// TIA Portal V21 export
FUNCTION "ZERO L" : Void   // FC10, LAD
{ S7_Optimized_Access := 'TRUE' }
// stored: SetENOAutomatically false
   VAR_TEMP
      "print ok" : String;
   END_VAR
   VAR_TEMP   // added for the SCL form of the ladder/FBD networks
      _w1 : Bool;
      _w2 : Bool;
      _w3 : Bool;
      _w4 : Bool;
      _w5 : Bool;
      _w6 : Bool;
      _w7 : Bool;
      _w8 : Bool;
      _w9 : Bool;
      _w10 : Bool;
      _w11 : Bool;
      _w12 : Bool;
   END_VAR
BEGIN

REGION Network 1
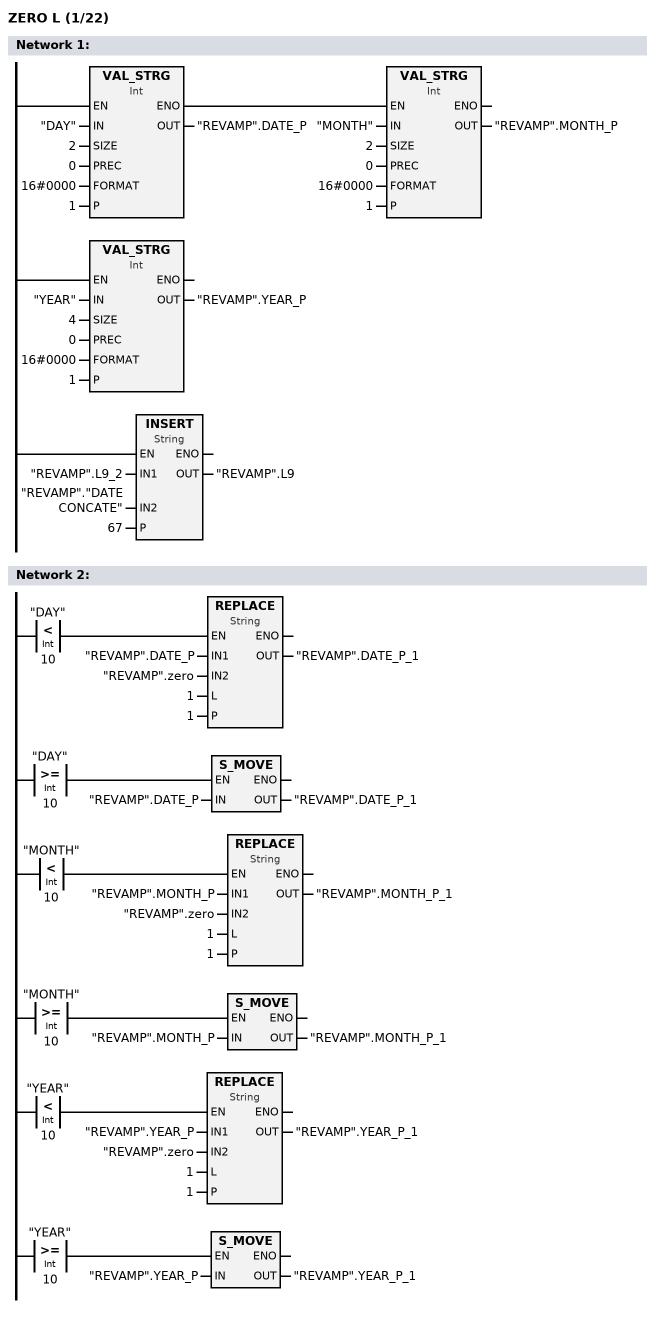
   RUNG wire#powerrail
      { S7_Templates := "[value_type := Int, str_type := String]" } VAL_STRG(IN := "DAY", SIZE := 2, PREC := 0, FORMAT := 16#0000, P := 1, OUT => "REVAMP".DATE_P)
      { S7_Templates := "[value_type := Int, str_type := String]" } VAL_STRG(IN := "MONTH", SIZE := 2, PREC := 0, FORMAT := 16#0000, P := 1, OUT => "REVAMP".MONTH_P)
   END_RUNG
   RUNG wire#powerrail
      { S7_Templates := "[value_type := Int, str_type := String]" } VAL_STRG(IN := "YEAR", SIZE := 4, PREC := 0, FORMAT := 16#0000, P := 1, OUT => "REVAMP".YEAR_P)
   END_RUNG
   RUNG wire#powerrail
      { S7_Templates := "str_type := String" } INSERT(IN1 := "REVAMP".L9_2, IN2 := "REVAMP"."DATE CONCATE", P := 67, OUT => "REVAMP".L9)
   END_RUNG
   // the same network as SCL:
   VAL_STRG(IN := "DAY", SIZE := 2, PREC := 0, FORMAT := 16#0000, P := 1, OUT => "REVAMP".DATE_P, ENO => #_w1);
   IF #_w1 THEN
       VAL_STRG(IN := "MONTH", SIZE := 2, PREC := 0, FORMAT := 16#0000, P := 1, OUT => "REVAMP".MONTH_P);
   END_IF;
   VAL_STRG(IN := "YEAR", SIZE := 4, PREC := 0, FORMAT := 16#0000, P := 1, OUT => "REVAMP".YEAR_P);
   INSERT(IN1 := "REVAMP".L9_2, IN2 := "REVAMP"."DATE CONCATE", P := 67, OUT => "REVAMP".L9);
END_REGION

REGION Network 2
   RUNG wire#powerrail
      { S7_Templates := "SrcType := Int" } LT_Contact(in1 := "DAY", in2 := 10)
      { S7_Templates := "str_type := String" } REPLACE(IN1 := "REVAMP".DATE_P, IN2 := "REVAMP".zero, L := 1, P := 1, OUT => "REVAMP".DATE_P_1)
   END_RUNG
   RUNG wire#powerrail
      { S7_Templates := "SrcType := Int" } GE_Contact(in1 := "DAY", in2 := 10)
      S_Move(in := "REVAMP".DATE_P, out => "REVAMP".DATE_P_1)
   END_RUNG
   RUNG wire#powerrail
      { S7_Templates := "SrcType := Int" } LT_Contact(in1 := "MONTH", in2 := 10)
      { S7_Templates := "str_type := String" } REPLACE(IN1 := "REVAMP".MONTH_P, IN2 := "REVAMP".zero, L := 1, P := 1, OUT => "REVAMP".MONTH_P_1)
   END_RUNG
   RUNG wire#powerrail
      { S7_Templates := "SrcType := Int" } GE_Contact(in1 := "MONTH", in2 := 10)
      S_Move(in := "REVAMP".MONTH_P, out => "REVAMP".MONTH_P_1)
   END_RUNG
   RUNG wire#powerrail
      { S7_Templates := "SrcType := Int" } LT_Contact(in1 := "YEAR", in2 := 10)
      { S7_Templates := "str_type := String" } REPLACE(IN1 := "REVAMP".YEAR_P, IN2 := "REVAMP".zero, L := 1, P := 1, OUT => "REVAMP".YEAR_P_1)
   END_RUNG
   RUNG wire#powerrail
      { S7_Templates := "SrcType := Int" } GE_Contact(in1 := "YEAR", in2 := 10)
      S_Move(in := "REVAMP".YEAR_P, out => "REVAMP".YEAR_P_1)
   END_RUNG
   // the same network as SCL:
   IF "DAY" < 10 THEN
       REPLACE(IN1 := "REVAMP".DATE_P, IN2 := "REVAMP".zero, L := 1, P := 1, OUT => "REVAMP".DATE_P_1);
   END_IF;
   IF "DAY" >= 10 THEN "REVAMP".DATE_P_1 := "REVAMP".DATE_P; END_IF;
   IF "MONTH" < 10 THEN
       REPLACE(IN1 := "REVAMP".MONTH_P, IN2 := "REVAMP".zero, L := 1, P := 1, OUT => "REVAMP".MONTH_P_1);
   END_IF;
   IF "MONTH" >= 10 THEN "REVAMP".MONTH_P_1 := "REVAMP".MONTH_P; END_IF;
   IF "YEAR" < 10 THEN
       REPLACE(IN1 := "REVAMP".YEAR_P, IN2 := "REVAMP".zero, L := 1, P := 1, OUT => "REVAMP".YEAR_P_1);
   END_IF;
   IF "YEAR" >= 10 THEN "REVAMP".YEAR_P_1 := "REVAMP".YEAR_P; END_IF;
END_REGION

REGION Network 3
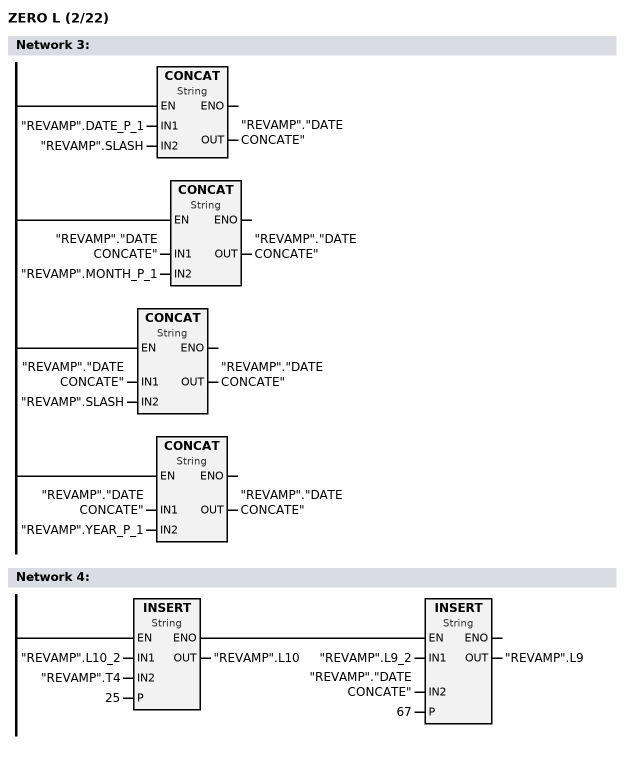
   RUNG wire#powerrail
      { S7_Templates := "[card := 2, str_type := String]" } CONCAT(IN1 := "REVAMP".DATE_P_1, IN2 := "REVAMP".SLASH, OUT => "REVAMP"."DATE CONCATE")
   END_RUNG
   RUNG wire#powerrail
      { S7_Templates := "[card := 2, str_type := String]" } CONCAT(IN1 := "REVAMP"."DATE CONCATE", IN2 := "REVAMP".MONTH_P_1, OUT => "REVAMP"."DATE CONCATE")
   END_RUNG
   RUNG wire#powerrail
      { S7_Templates := "[card := 2, str_type := String]" } CONCAT(IN1 := "REVAMP"."DATE CONCATE", IN2 := "REVAMP".SLASH, OUT => "REVAMP"."DATE CONCATE")
   END_RUNG
   RUNG wire#powerrail
      { S7_Templates := "[card := 2, str_type := String]" } CONCAT(IN1 := "REVAMP"."DATE CONCATE", IN2 := "REVAMP".YEAR_P_1, OUT => "REVAMP"."DATE CONCATE")
   END_RUNG
   // the same network as SCL:
   CONCAT(IN1 := "REVAMP".DATE_P_1, IN2 := "REVAMP".SLASH, OUT => "REVAMP"."DATE CONCATE");
   CONCAT(IN1 := "REVAMP"."DATE CONCATE", IN2 := "REVAMP".MONTH_P_1, OUT => "REVAMP"."DATE CONCATE");
   CONCAT(IN1 := "REVAMP"."DATE CONCATE", IN2 := "REVAMP".SLASH, OUT => "REVAMP"."DATE CONCATE");
   CONCAT(IN1 := "REVAMP"."DATE CONCATE", IN2 := "REVAMP".YEAR_P_1, OUT => "REVAMP"."DATE CONCATE");
END_REGION

REGION Network 4
   RUNG wire#powerrail
      { S7_Templates := "str_type := String" } INSERT(IN1 := "REVAMP".L10_2, IN2 := "REVAMP".T4, P := 25, OUT => "REVAMP".L10)
      { S7_Templates := "str_type := String" } INSERT(IN1 := "REVAMP".L9_2, IN2 := "REVAMP"."DATE CONCATE", P := 67, OUT => "REVAMP".L9)
   END_RUNG
   // the same network as SCL:
   INSERT(IN1 := "REVAMP".L10_2, IN2 := "REVAMP".T4, P := 25, OUT => "REVAMP".L10, ENO => #_w1);
   IF #_w1 THEN
       INSERT(IN1 := "REVAMP".L9_2, IN2 := "REVAMP"."DATE CONCATE", P := 67, OUT => "REVAMP".L9);
   END_IF;
END_REGION

REGION Network 5
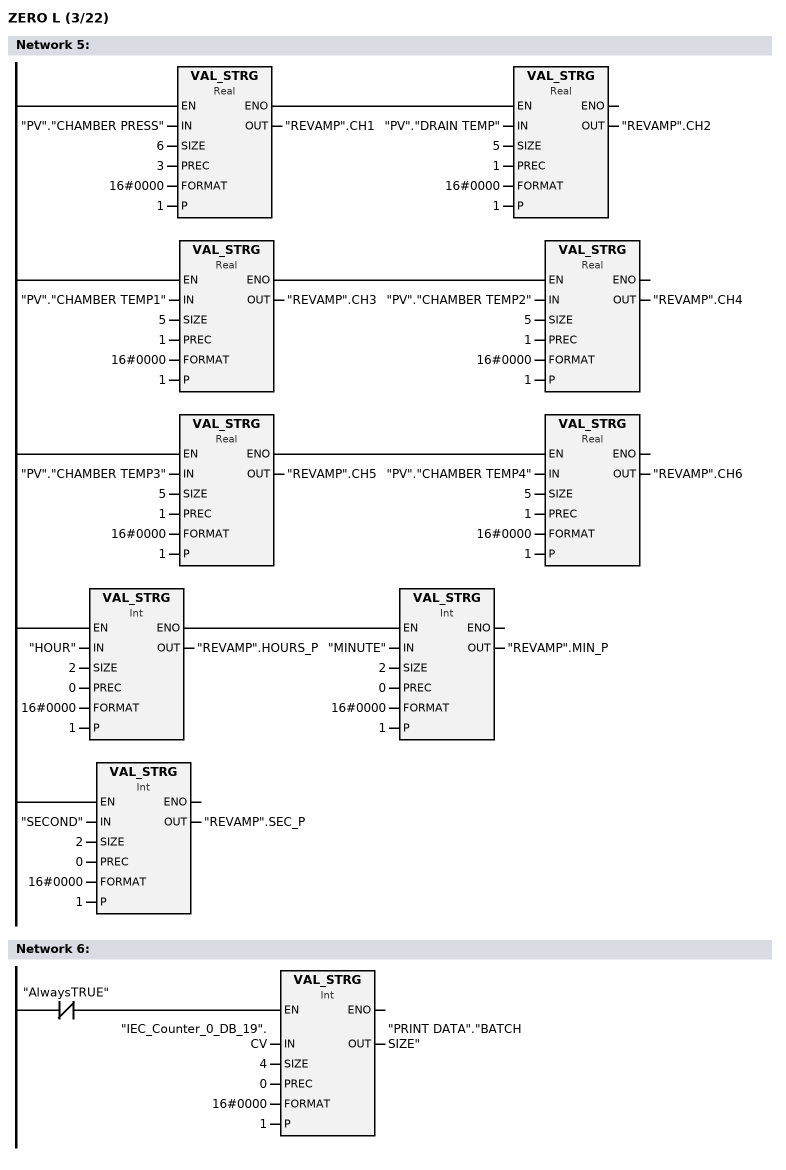
   RUNG wire#powerrail
      { S7_Templates := "[value_type := Real, str_type := String]" } VAL_STRG(IN := "PV"."CHAMBER PRESS", SIZE := 6, PREC := 3, FORMAT := 16#0000, P := 1, OUT => "REVAMP".CH1)
      { S7_Templates := "[value_type := Real, str_type := String]" } VAL_STRG(IN := "PV"."DRAIN TEMP", SIZE := 5, PREC := 1, FORMAT := 16#0000, P := 1, OUT => "REVAMP".CH2)
   END_RUNG
   RUNG wire#powerrail
      { S7_Templates := "[value_type := Real, str_type := String]" } VAL_STRG(IN := "PV"."CHAMBER TEMP1", SIZE := 5, PREC := 1, FORMAT := 16#0000, P := 1, OUT => "REVAMP".CH3)
      { S7_Templates := "[value_type := Real, str_type := String]" } VAL_STRG(IN := "PV"."CHAMBER TEMP2", SIZE := 5, PREC := 1, FORMAT := 16#0000, P := 1, OUT => "REVAMP".CH4)
   END_RUNG
   RUNG wire#powerrail
      { S7_Templates := "[value_type := Real, str_type := String]" } VAL_STRG(IN := "PV"."CHAMBER TEMP3", SIZE := 5, PREC := 1, FORMAT := 16#0000, P := 1, OUT => "REVAMP".CH5)
      { S7_Templates := "[value_type := Real, str_type := String]" } VAL_STRG(IN := "PV"."CHAMBER TEMP4", SIZE := 5, PREC := 1, FORMAT := 16#0000, P := 1, OUT => "REVAMP".CH6)
   END_RUNG
   RUNG wire#powerrail
      { S7_Templates := "[value_type := Int, str_type := String]" } VAL_STRG(IN := "HOUR", SIZE := 2, PREC := 0, FORMAT := 16#0000, P := 1, OUT => "REVAMP".HOURS_P)
      { S7_Templates := "[value_type := Int, str_type := String]" } VAL_STRG(IN := "MINUTE", SIZE := 2, PREC := 0, FORMAT := 16#0000, P := 1, OUT => "REVAMP".MIN_P)
   END_RUNG
   RUNG wire#powerrail
      { S7_Templates := "[value_type := Int, str_type := String]" } VAL_STRG(IN := "SECOND", SIZE := 2, PREC := 0, FORMAT := 16#0000, P := 1, OUT => "REVAMP".SEC_P)
   END_RUNG
   // the same network as SCL:
   VAL_STRG(IN := "PV"."CHAMBER PRESS",
            SIZE := 6,
            PREC := 3,
            FORMAT := 16#0000,
            P := 1,
            OUT => "REVAMP".CH1,
            ENO => #_w1);
   IF #_w1 THEN
       VAL_STRG(IN := "PV"."DRAIN TEMP", SIZE := 5, PREC := 1, FORMAT := 16#0000, P := 1, OUT => "REVAMP".CH2);
   END_IF;
   VAL_STRG(IN := "PV"."CHAMBER TEMP1",
            SIZE := 5,
            PREC := 1,
            FORMAT := 16#0000,
            P := 1,
            OUT => "REVAMP".CH3,
            ENO => #_w2);
   IF #_w2 THEN
       VAL_STRG(IN := "PV"."CHAMBER TEMP2", SIZE := 5, PREC := 1, FORMAT := 16#0000, P := 1, OUT => "REVAMP".CH4);
   END_IF;
   VAL_STRG(IN := "PV"."CHAMBER TEMP3",
            SIZE := 5,
            PREC := 1,
            FORMAT := 16#0000,
            P := 1,
            OUT => "REVAMP".CH5,
            ENO => #_w3);
   IF #_w3 THEN
       VAL_STRG(IN := "PV"."CHAMBER TEMP4", SIZE := 5, PREC := 1, FORMAT := 16#0000, P := 1, OUT => "REVAMP".CH6);
   END_IF;
   VAL_STRG(IN := "HOUR", SIZE := 2, PREC := 0, FORMAT := 16#0000, P := 1, OUT => "REVAMP".HOURS_P, ENO => #_w4);
   IF #_w4 THEN
       VAL_STRG(IN := "MINUTE", SIZE := 2, PREC := 0, FORMAT := 16#0000, P := 1, OUT => "REVAMP".MIN_P);
   END_IF;
   VAL_STRG(IN := "SECOND", SIZE := 2, PREC := 0, FORMAT := 16#0000, P := 1, OUT => "REVAMP".SEC_P);
END_REGION

REGION Network 6
   RUNG wire#powerrail
      I_Contact( "AlwaysTRUE" )
      { S7_Templates := "[value_type := Int, str_type := String]" } VAL_STRG(IN := "IEC_Counter_0_DB_19".CV, SIZE := 4, PREC := 0, FORMAT := 16#0000, P := 1, OUT => "PRINT DATA"."BATCH SIZE")
   END_RUNG
   // the same network as SCL:
   IF NOT "AlwaysTRUE" THEN
       VAL_STRG(IN := "IEC_Counter_0_DB_19".CV,
                SIZE := 4,
                PREC := 0,
                FORMAT := 16#0000,
                P := 1,
                OUT => "PRINT DATA"."BATCH SIZE");
   END_IF;
END_REGION

REGION Network 7
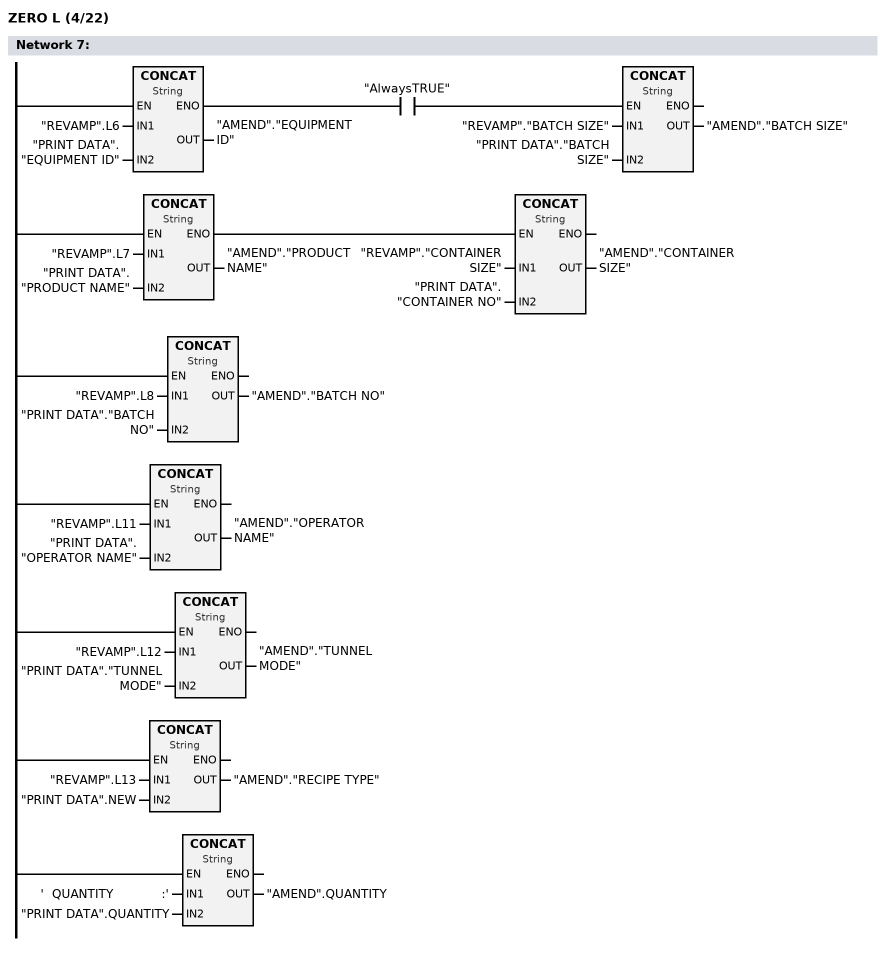
   RUNG wire#powerrail
      { S7_Templates := "[card := 2, str_type := String]" } CONCAT(IN1 := "REVAMP".L6, IN2 := "PRINT DATA"."EQUIPMENT ID", OUT => "AMEND"."EQUIPMENT ID")
      Contact( "AlwaysTRUE" )
      { S7_Templates := "[card := 2, str_type := String]" } CONCAT(IN1 := "REVAMP"."BATCH SIZE", IN2 := "PRINT DATA"."BATCH SIZE", OUT => "AMEND"."BATCH SIZE")
   END_RUNG
   RUNG wire#powerrail
      { S7_Templates := "[card := 2, str_type := String]" } CONCAT(IN1 := "REVAMP".L7, IN2 := "PRINT DATA"."PRODUCT NAME", OUT => "AMEND"."PRODUCT NAME")
      { S7_Templates := "[card := 2, str_type := String]" } CONCAT(IN1 := "REVAMP"."CONTAINER SIZE", IN2 := "PRINT DATA"."CONTAINER NO", OUT => "AMEND"."CONTAINER SIZE")
   END_RUNG
   RUNG wire#powerrail
      { S7_Templates := "[card := 2, str_type := String]" } CONCAT(IN1 := "REVAMP".L8, IN2 := "PRINT DATA"."BATCH NO", OUT => "AMEND"."BATCH NO")
   END_RUNG
   RUNG wire#powerrail
      { S7_Templates := "[card := 2, str_type := String]" } CONCAT(IN1 := "REVAMP".L11, IN2 := "PRINT DATA"."OPERATOR NAME", OUT => "AMEND"."OPERATOR NAME")
   END_RUNG
   RUNG wire#powerrail
      { S7_Templates := "[card := 2, str_type := String]" } CONCAT(IN1 := "REVAMP".L12, IN2 := "PRINT DATA"."TUNNEL MODE", OUT => "AMEND"."TUNNEL MODE")
   END_RUNG
   RUNG wire#powerrail
      { S7_Templates := "[card := 2, str_type := String]" } CONCAT(IN1 := "REVAMP".L13, IN2 := "PRINT DATA".NEW, OUT => "AMEND"."RECIPE TYPE")
   END_RUNG
   RUNG wire#powerrail
      { S7_Templates := "[card := 2, str_type := String]" } CONCAT(IN1 := '  QUANTITY            :', IN2 := "PRINT DATA".QUANTITY, OUT => "AMEND".QUANTITY)
   END_RUNG
   // the same network as SCL:
   CONCAT(IN1 := "REVAMP".L6, IN2 := "PRINT DATA"."EQUIPMENT ID", OUT => "AMEND"."EQUIPMENT ID", ENO => #_w1);
   IF #_w1 AND "AlwaysTRUE" THEN
       CONCAT(IN1 := "REVAMP"."BATCH SIZE", IN2 := "PRINT DATA"."BATCH SIZE", OUT => "AMEND"."BATCH SIZE");
   END_IF;
   CONCAT(IN1 := "REVAMP".L7, IN2 := "PRINT DATA"."PRODUCT NAME", OUT => "AMEND"."PRODUCT NAME", ENO => #_w2);
   IF #_w2 THEN
       CONCAT(IN1 := "REVAMP"."CONTAINER SIZE", IN2 := "PRINT DATA"."CONTAINER NO", OUT => "AMEND"."CONTAINER SIZE");
   END_IF;
   CONCAT(IN1 := "REVAMP".L8, IN2 := "PRINT DATA"."BATCH NO", OUT => "AMEND"."BATCH NO");
   CONCAT(IN1 := "REVAMP".L11, IN2 := "PRINT DATA"."OPERATOR NAME", OUT => "AMEND"."OPERATOR NAME");
   CONCAT(IN1 := "REVAMP".L12, IN2 := "PRINT DATA"."TUNNEL MODE", OUT => "AMEND"."TUNNEL MODE");
   CONCAT(IN1 := "REVAMP".L13, IN2 := "PRINT DATA".NEW, OUT => "AMEND"."RECIPE TYPE");
   CONCAT(IN1 := '  QUANTITY            :', IN2 := "PRINT DATA".QUANTITY, OUT => "AMEND".QUANTITY);
END_REGION

REGION Network 8
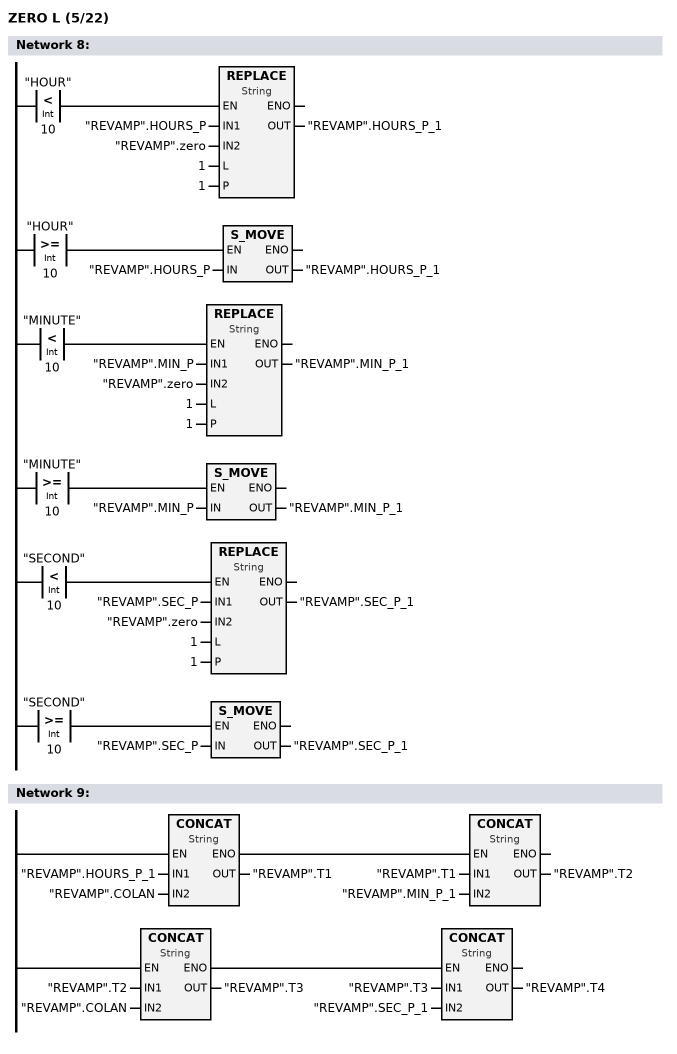
   RUNG wire#powerrail
      { S7_Templates := "SrcType := Int" } LT_Contact(in1 := "HOUR", in2 := 10)
      { S7_Templates := "str_type := String" } REPLACE(IN1 := "REVAMP".HOURS_P, IN2 := "REVAMP".zero, L := 1, P := 1, OUT => "REVAMP".HOURS_P_1)
   END_RUNG
   RUNG wire#powerrail
      { S7_Templates := "SrcType := Int" } GE_Contact(in1 := "HOUR", in2 := 10)
      S_Move(in := "REVAMP".HOURS_P, out => "REVAMP".HOURS_P_1)
   END_RUNG
   RUNG wire#powerrail
      { S7_Templates := "SrcType := Int" } LT_Contact(in1 := "MINUTE", in2 := 10)
      { S7_Templates := "str_type := String" } REPLACE(IN1 := "REVAMP".MIN_P, IN2 := "REVAMP".zero, L := 1, P := 1, OUT => "REVAMP".MIN_P_1)
   END_RUNG
   RUNG wire#powerrail
      { S7_Templates := "SrcType := Int" } GE_Contact(in1 := "MINUTE", in2 := 10)
      S_Move(in := "REVAMP".MIN_P, out => "REVAMP".MIN_P_1)
   END_RUNG
   RUNG wire#powerrail
      { S7_Templates := "SrcType := Int" } LT_Contact(in1 := "SECOND", in2 := 10)
      { S7_Templates := "str_type := String" } REPLACE(IN1 := "REVAMP".SEC_P, IN2 := "REVAMP".zero, L := 1, P := 1, OUT => "REVAMP".SEC_P_1)
   END_RUNG
   RUNG wire#powerrail
      { S7_Templates := "SrcType := Int" } GE_Contact(in1 := "SECOND", in2 := 10)
      S_Move(in := "REVAMP".SEC_P, out => "REVAMP".SEC_P_1)
   END_RUNG
   // the same network as SCL:
   IF "HOUR" < 10 THEN
       REPLACE(IN1 := "REVAMP".HOURS_P, IN2 := "REVAMP".zero, L := 1, P := 1, OUT => "REVAMP".HOURS_P_1);
   END_IF;
   IF "HOUR" >= 10 THEN "REVAMP".HOURS_P_1 := "REVAMP".HOURS_P; END_IF;
   IF "MINUTE" < 10 THEN
       REPLACE(IN1 := "REVAMP".MIN_P, IN2 := "REVAMP".zero, L := 1, P := 1, OUT => "REVAMP".MIN_P_1);
   END_IF;
   IF "MINUTE" >= 10 THEN "REVAMP".MIN_P_1 := "REVAMP".MIN_P; END_IF;
   IF "SECOND" < 10 THEN
       REPLACE(IN1 := "REVAMP".SEC_P, IN2 := "REVAMP".zero, L := 1, P := 1, OUT => "REVAMP".SEC_P_1);
   END_IF;
   IF "SECOND" >= 10 THEN "REVAMP".SEC_P_1 := "REVAMP".SEC_P; END_IF;
END_REGION

REGION Network 9
   RUNG wire#powerrail
      { S7_Templates := "[card := 2, str_type := String]" } CONCAT(IN1 := "REVAMP".HOURS_P_1, IN2 := "REVAMP".COLAN, OUT => "REVAMP".T1)
      { S7_Templates := "[card := 2, str_type := String]" } CONCAT(IN1 := "REVAMP".T1, IN2 := "REVAMP".MIN_P_1, OUT => "REVAMP".T2)
   END_RUNG
   RUNG wire#powerrail
      { S7_Templates := "[card := 2, str_type := String]" } CONCAT(IN1 := "REVAMP".T2, IN2 := "REVAMP".COLAN, OUT => "REVAMP".T3)
      { S7_Templates := "[card := 2, str_type := String]" } CONCAT(IN1 := "REVAMP".T3, IN2 := "REVAMP".SEC_P_1, OUT => "REVAMP".T4)
   END_RUNG
   // the same network as SCL:
   CONCAT(IN1 := "REVAMP".HOURS_P_1, IN2 := "REVAMP".COLAN, OUT => "REVAMP".T1, ENO => #_w1);
   IF #_w1 THEN CONCAT(IN1 := "REVAMP".T1, IN2 := "REVAMP".MIN_P_1, OUT => "REVAMP".T2); END_IF;
   CONCAT(IN1 := "REVAMP".T2, IN2 := "REVAMP".COLAN, OUT => "REVAMP".T3, ENO => #_w2);
   IF #_w2 THEN CONCAT(IN1 := "REVAMP".T3, IN2 := "REVAMP".SEC_P_1, OUT => "REVAMP".T4); END_IF;
END_REGION

REGION Network 10
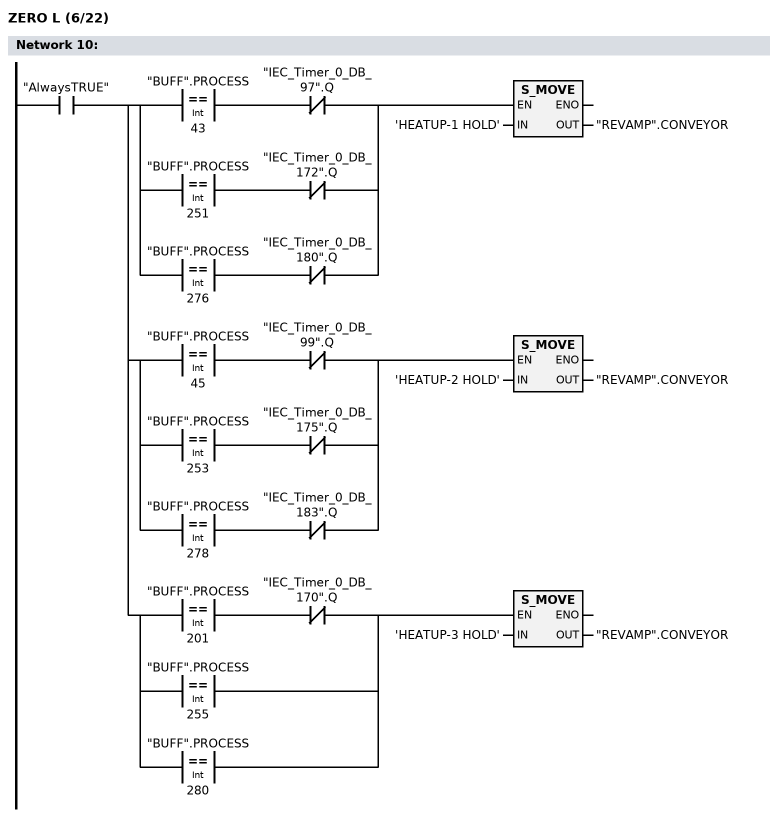
   RUNG wire#powerrail
      Contact( "AlwaysTRUE" )
      wire#w1
      { S7_Templates := "SrcType := Int" } EQ_Contact(in1 := "BUFF".PROCESS, in2 := 43)
      I_Contact( "IEC_Timer_0_DB_97".Q )
      wire#w2
      S_Move(in := 'HEATUP-1 HOLD', out => "REVAMP".CONVEYOR)
   END_RUNG
   RUNG wire#w1
      { S7_Templates := "SrcType := Int" } EQ_Contact(in1 := "BUFF".PROCESS, in2 := 251)
      I_Contact( "IEC_Timer_0_DB_172".Q )
   END_RUNG wire#w2
   RUNG wire#w1
      { S7_Templates := "SrcType := Int" } EQ_Contact(in1 := "BUFF".PROCESS, in2 := 276)
      I_Contact( "IEC_Timer_0_DB_180".Q )
   END_RUNG wire#w2
   RUNG wire#w1
      { S7_Templates := "SrcType := Int" } EQ_Contact(in1 := "BUFF".PROCESS, in2 := 45)
      I_Contact( "IEC_Timer_0_DB_99".Q )
      wire#w3
      S_Move(in := 'HEATUP-2 HOLD', out => "REVAMP".CONVEYOR)
   END_RUNG
   RUNG wire#w1
      { S7_Templates := "SrcType := Int" } EQ_Contact(in1 := "BUFF".PROCESS, in2 := 253)
      I_Contact( "IEC_Timer_0_DB_175".Q )
   END_RUNG wire#w3
   RUNG wire#w1
      { S7_Templates := "SrcType := Int" } EQ_Contact(in1 := "BUFF".PROCESS, in2 := 278)
      I_Contact( "IEC_Timer_0_DB_183".Q )
   END_RUNG wire#w3
   RUNG wire#w1
      { S7_Templates := "SrcType := Int" } EQ_Contact(in1 := "BUFF".PROCESS, in2 := 201)
      I_Contact( "IEC_Timer_0_DB_170".Q )
      wire#w4
      S_Move(in := 'HEATUP-3 HOLD', out => "REVAMP".CONVEYOR)
   END_RUNG
   RUNG wire#w1
      { S7_Templates := "SrcType := Int" } EQ_Contact(in1 := "BUFF".PROCESS, in2 := 255)
   END_RUNG wire#w4
   RUNG wire#w1
      { S7_Templates := "SrcType := Int" } EQ_Contact(in1 := "BUFF".PROCESS, in2 := 280)
   END_RUNG wire#w4
   // the same network as SCL:
   IF "AlwaysTRUE" AND ((("BUFF".PROCESS = 43) AND NOT "IEC_Timer_0_DB_97".Q) OR (("BUFF".PROCESS = 251) AND NOT "IEC_Timer_0_DB_172".Q) OR (("BUFF".PROCESS = 276) AND NOT "IEC_Timer_0_DB_180".Q)) THEN
       "REVAMP".CONVEYOR := 'HEATUP-1 HOLD';
   END_IF;
   IF "AlwaysTRUE" AND ((("BUFF".PROCESS = 45) AND NOT "IEC_Timer_0_DB_99".Q) OR (("BUFF".PROCESS = 253) AND NOT "IEC_Timer_0_DB_175".Q) OR (("BUFF".PROCESS = 278) AND NOT "IEC_Timer_0_DB_183".Q)) THEN
       "REVAMP".CONVEYOR := 'HEATUP-2 HOLD';
   END_IF;
   IF "AlwaysTRUE" AND ((("BUFF".PROCESS = 201) AND NOT "IEC_Timer_0_DB_170".Q) OR ("BUFF".PROCESS = 255) OR ("BUFF".PROCESS = 280)) THEN
       "REVAMP".CONVEYOR := 'HEATUP-3 HOLD';
   END_IF;
END_REGION

REGION Network 11
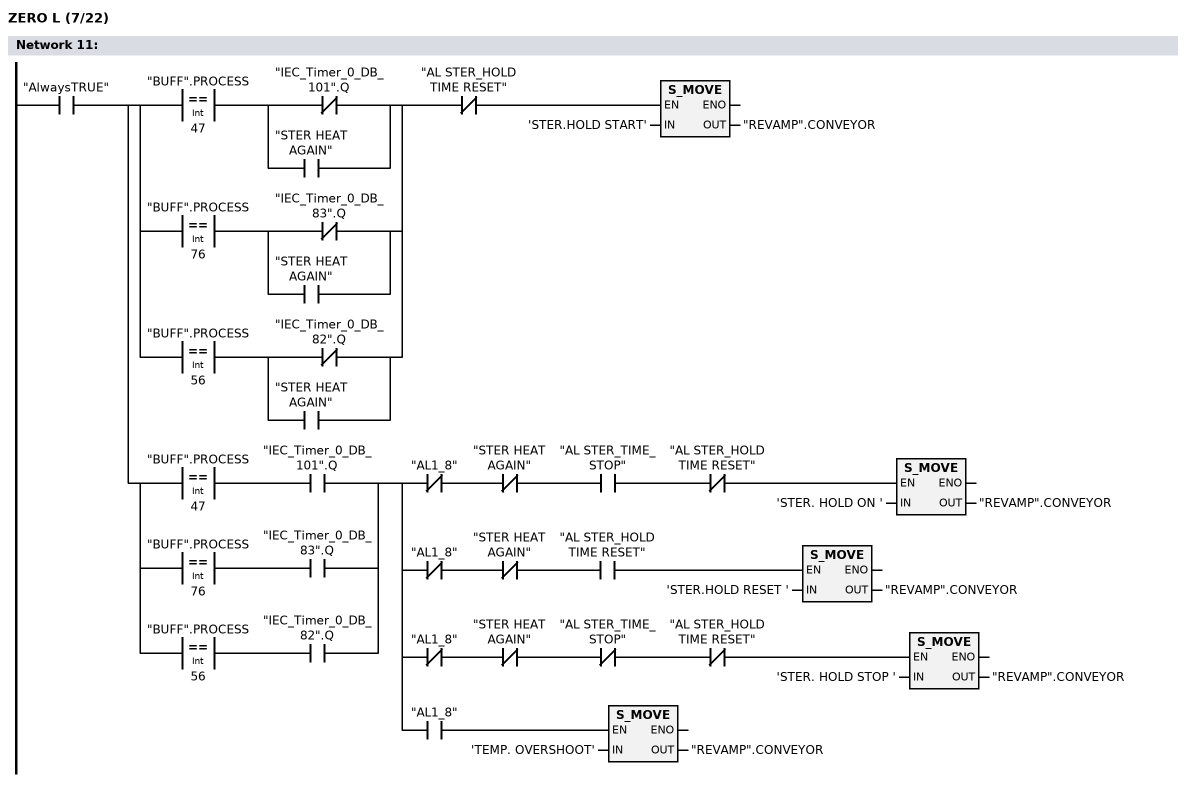
   RUNG wire#powerrail
      Contact( "AlwaysTRUE" )
      wire#w1
      { S7_Templates := "SrcType := Int" } EQ_Contact(in1 := "BUFF".PROCESS, in2 := 47)
      wire#w2
      I_Contact( "IEC_Timer_0_DB_101".Q )
      wire#w3
      I_Contact( "AL STER_HOLD TIME RESET" )
      S_Move(in := 'STER.HOLD START', out => "REVAMP".CONVEYOR)
   END_RUNG
   RUNG wire#w2
      Contact( "STER HEAT AGAIN" )
   END_RUNG wire#w3
   RUNG wire#w1
      { S7_Templates := "SrcType := Int" } EQ_Contact(in1 := "BUFF".PROCESS, in2 := 76)
      wire#w4
      I_Contact( "IEC_Timer_0_DB_83".Q )
   END_RUNG wire#w3
   RUNG wire#w4
      Contact( "STER HEAT AGAIN" )
   END_RUNG wire#w3
   RUNG wire#w1
      { S7_Templates := "SrcType := Int" } EQ_Contact(in1 := "BUFF".PROCESS, in2 := 56)
      wire#w5
      I_Contact( "IEC_Timer_0_DB_82".Q )
   END_RUNG wire#w3
   RUNG wire#w5
      Contact( "STER HEAT AGAIN" )
   END_RUNG wire#w3
   RUNG wire#w1
      { S7_Templates := "SrcType := Int" } EQ_Contact(in1 := "BUFF".PROCESS, in2 := 47)
      Contact( "IEC_Timer_0_DB_101".Q )
      wire#w6
      I_Contact( "AL1_8" )
      I_Contact( "STER HEAT AGAIN" )
      Contact( "AL STER_TIME_STOP" )
      I_Contact( "AL STER_HOLD TIME RESET" )
      S_Move(in := 'STER. HOLD ON ', out => "REVAMP".CONVEYOR)
   END_RUNG
   RUNG wire#w1
      { S7_Templates := "SrcType := Int" } EQ_Contact(in1 := "BUFF".PROCESS, in2 := 76)
      Contact( "IEC_Timer_0_DB_83".Q )
   END_RUNG wire#w6
   RUNG wire#w1
      { S7_Templates := "SrcType := Int" } EQ_Contact(in1 := "BUFF".PROCESS, in2 := 56)
      Contact( "IEC_Timer_0_DB_82".Q )
   END_RUNG wire#w6
   RUNG wire#w6
      I_Contact( "AL1_8" )
      I_Contact( "STER HEAT AGAIN" )
      Contact( "AL STER_HOLD TIME RESET" )
      S_Move(in := 'STER.HOLD RESET ', out => "REVAMP".CONVEYOR)
   END_RUNG
   RUNG wire#w6
      I_Contact( "AL1_8" )
      I_Contact( "STER HEAT AGAIN" )
      I_Contact( "AL STER_TIME_STOP" )
      I_Contact( "AL STER_HOLD TIME RESET" )
      S_Move(in := 'STER. HOLD STOP ', out => "REVAMP".CONVEYOR)
   END_RUNG
   RUNG wire#w6
      Contact( "AL1_8" )
      S_Move(in := 'TEMP. OVERSHOOT', out => "REVAMP".CONVEYOR)
   END_RUNG
   // the same network as SCL:
   IF "AlwaysTRUE" AND ((("BUFF".PROCESS = 47) AND (NOT "IEC_Timer_0_DB_101".Q OR "STER HEAT AGAIN")) OR (("BUFF".PROCESS = 76) AND (NOT "IEC_Timer_0_DB_83".Q OR "STER HEAT AGAIN")) OR (("BUFF".PROCESS = 56) AND (NOT "IEC_Timer_0_DB_82".Q OR "STER HEAT AGAIN"))) AND NOT "AL STER_HOLD TIME RESET" THEN
       "REVAMP".CONVEYOR := 'STER.HOLD START';
   END_IF;
   #_w1 := "AlwaysTRUE" AND ((("BUFF".PROCESS = 47) AND "IEC_Timer_0_DB_101".Q) OR (("BUFF".PROCESS = 76) AND "IEC_Timer_0_DB_83".Q) OR (("BUFF".PROCESS = 56) AND "IEC_Timer_0_DB_82".Q));
   IF #_w1 AND NOT "AL1_8" AND NOT "STER HEAT AGAIN" AND "AL STER_TIME_STOP" AND NOT "AL STER_HOLD TIME RESET" THEN
       "REVAMP".CONVEYOR := 'STER. HOLD ON ';
   END_IF;
   IF #_w1 AND NOT "AL1_8" AND NOT "STER HEAT AGAIN" AND "AL STER_HOLD TIME RESET" THEN
       "REVAMP".CONVEYOR := 'STER.HOLD RESET ';
   END_IF;
   IF #_w1 AND NOT "AL1_8" AND NOT "STER HEAT AGAIN" AND NOT "AL STER_TIME_STOP" AND NOT "AL STER_HOLD TIME RESET" THEN
       "REVAMP".CONVEYOR := 'STER. HOLD STOP ';
   END_IF;
   IF #_w1 AND "AL1_8" THEN "REVAMP".CONVEYOR := 'TEMP. OVERSHOOT'; END_IF;
END_REGION

REGION Network 12
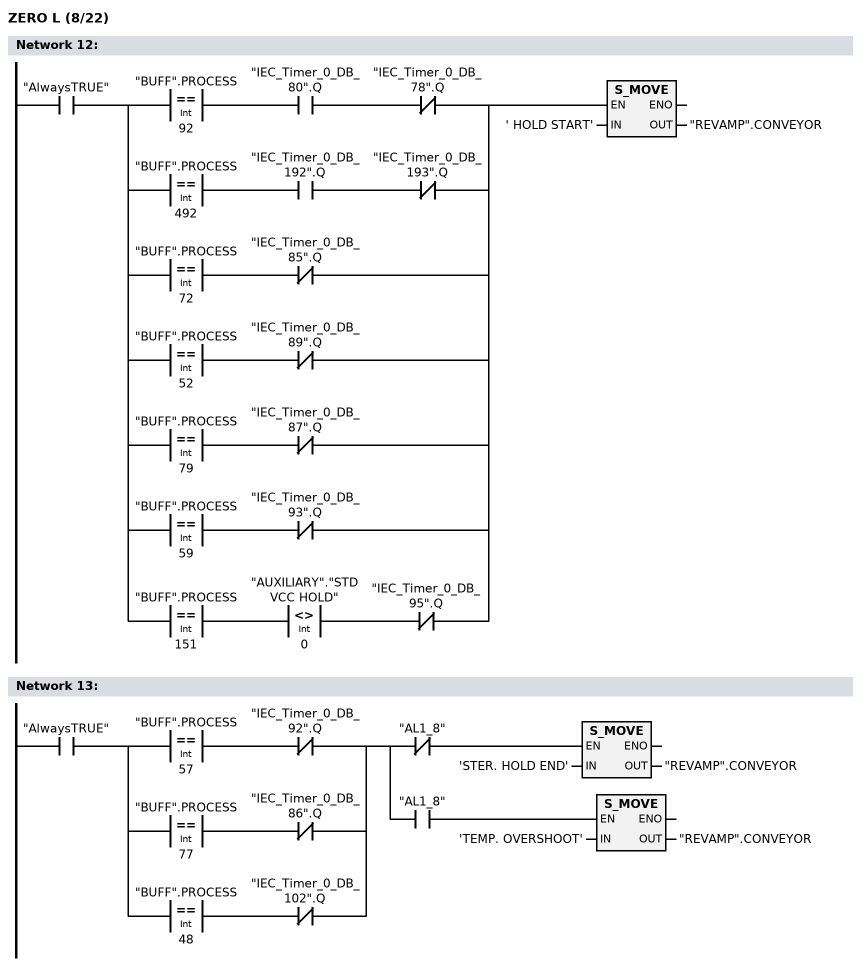
   RUNG wire#powerrail
      Contact( "AlwaysTRUE" )
      wire#w1
      { S7_Templates := "SrcType := Int" } EQ_Contact(in1 := "BUFF".PROCESS, in2 := 92)
      Contact( "IEC_Timer_0_DB_80".Q )
      I_Contact( "IEC_Timer_0_DB_78".Q )
      wire#w2
      S_Move(in := ' HOLD START', out => "REVAMP".CONVEYOR)
   END_RUNG
   RUNG wire#w1
      { S7_Templates := "SrcType := Int" } EQ_Contact(in1 := "BUFF".PROCESS, in2 := 492)
      Contact( "IEC_Timer_0_DB_192".Q )
      I_Contact( "IEC_Timer_0_DB_193".Q )
   END_RUNG wire#w2
   RUNG wire#w1
      { S7_Templates := "SrcType := Int" } EQ_Contact(in1 := "BUFF".PROCESS, in2 := 72)
      I_Contact( "IEC_Timer_0_DB_85".Q )
   END_RUNG wire#w2
   RUNG wire#w1
      { S7_Templates := "SrcType := Int" } EQ_Contact(in1 := "BUFF".PROCESS, in2 := 52)
      I_Contact( "IEC_Timer_0_DB_89".Q )
   END_RUNG wire#w2
   RUNG wire#w1
      { S7_Templates := "SrcType := Int" } EQ_Contact(in1 := "BUFF".PROCESS, in2 := 79)
      I_Contact( "IEC_Timer_0_DB_87".Q )
   END_RUNG wire#w2
   RUNG wire#w1
      { S7_Templates := "SrcType := Int" } EQ_Contact(in1 := "BUFF".PROCESS, in2 := 59)
      I_Contact( "IEC_Timer_0_DB_93".Q )
   END_RUNG wire#w2
   RUNG wire#w1
      { S7_Templates := "SrcType := Int" } EQ_Contact(in1 := "BUFF".PROCESS, in2 := 151)
      { S7_Templates := "SrcType := Int" } NE_Contact(in1 := "AUXILIARY"."STD VCC HOLD", in2 := 0)
      I_Contact( "IEC_Timer_0_DB_95".Q )
   END_RUNG wire#w2
   // the same network as SCL:
   IF "AlwaysTRUE" AND ((("BUFF".PROCESS = 92) AND "IEC_Timer_0_DB_80".Q AND NOT "IEC_Timer_0_DB_78".Q) OR (("BUFF".PROCESS = 492) AND "IEC_Timer_0_DB_192".Q AND NOT "IEC_Timer_0_DB_193".Q) OR (("BUFF".PROCESS = 72) AND NOT "IEC_Timer_0_DB_85".Q) OR (("BUFF".PROCESS = 52) AND NOT "IEC_Timer_0_DB_89".Q) OR (("BUFF".PROCESS = 79) AND NOT "IEC_Timer_0_DB_87".Q) OR (("BUFF".PROCESS = 59) AND NOT "IEC_Timer_0_DB_93".Q) OR (("BUFF".PROCESS = 151) AND ("AUXILIARY"."STD VCC HOLD" <> 0) AND NOT "IEC_Timer_0_DB_95".Q)) THEN
       "REVAMP".CONVEYOR := ' HOLD START';
   END_IF;
END_REGION

REGION Network 13
   RUNG wire#powerrail
      Contact( "AlwaysTRUE" )
      wire#w1
      { S7_Templates := "SrcType := Int" } EQ_Contact(in1 := "BUFF".PROCESS, in2 := 57)
      I_Contact( "IEC_Timer_0_DB_92".Q )
      wire#w2
      I_Contact( "AL1_8" )
      S_Move(in := 'STER. HOLD END', out => "REVAMP".CONVEYOR)
   END_RUNG
   RUNG wire#w1
      { S7_Templates := "SrcType := Int" } EQ_Contact(in1 := "BUFF".PROCESS, in2 := 77)
      I_Contact( "IEC_Timer_0_DB_86".Q )
   END_RUNG wire#w2
   RUNG wire#w1
      { S7_Templates := "SrcType := Int" } EQ_Contact(in1 := "BUFF".PROCESS, in2 := 48)
      I_Contact( "IEC_Timer_0_DB_102".Q )
   END_RUNG wire#w2
   RUNG wire#w2
      Contact( "AL1_8" )
      S_Move(in := 'TEMP. OVERSHOOT', out => "REVAMP".CONVEYOR)
   END_RUNG
   // the same network as SCL:
   #_w1 := "AlwaysTRUE" AND ((("BUFF".PROCESS = 57) AND NOT "IEC_Timer_0_DB_92".Q) OR (("BUFF".PROCESS = 77) AND NOT "IEC_Timer_0_DB_86".Q) OR (("BUFF".PROCESS = 48) AND NOT "IEC_Timer_0_DB_102".Q));
   IF #_w1 AND NOT "AL1_8" THEN "REVAMP".CONVEYOR := 'STER. HOLD END'; END_IF;
   IF #_w1 AND "AL1_8" THEN "REVAMP".CONVEYOR := 'TEMP. OVERSHOOT'; END_IF;
END_REGION

REGION Network 14
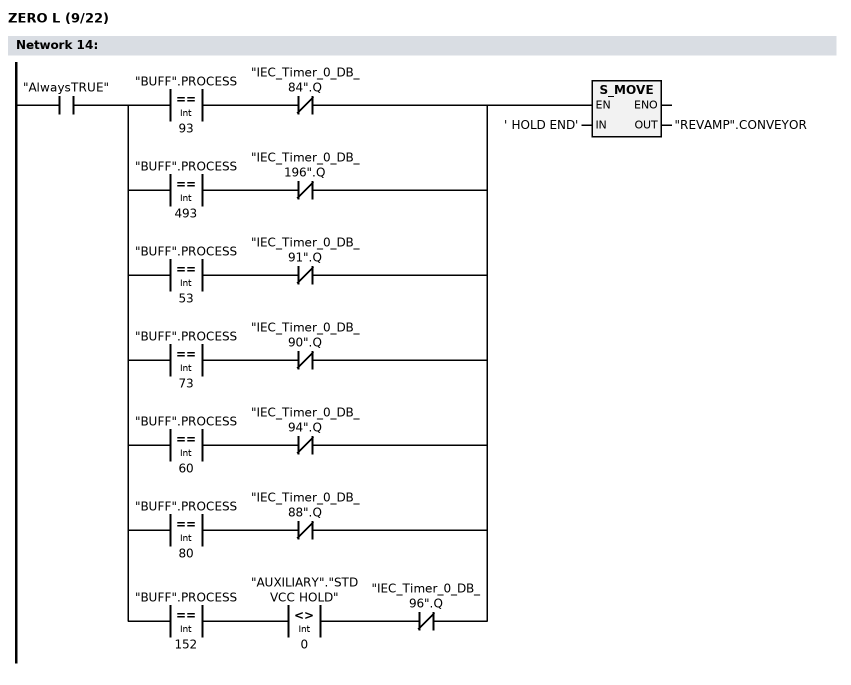
   RUNG wire#powerrail
      Contact( "AlwaysTRUE" )
      wire#w1
      { S7_Templates := "SrcType := Int" } EQ_Contact(in1 := "BUFF".PROCESS, in2 := 93)
      I_Contact( "IEC_Timer_0_DB_84".Q )
      wire#w2
      S_Move(in := ' HOLD END', out => "REVAMP".CONVEYOR)
   END_RUNG
   RUNG wire#w1
      { S7_Templates := "SrcType := Int" } EQ_Contact(in1 := "BUFF".PROCESS, in2 := 493)
      I_Contact( "IEC_Timer_0_DB_196".Q )
   END_RUNG wire#w2
   RUNG wire#w1
      { S7_Templates := "SrcType := Int" } EQ_Contact(in1 := "BUFF".PROCESS, in2 := 53)
      I_Contact( "IEC_Timer_0_DB_91".Q )
   END_RUNG wire#w2
   RUNG wire#w1
      { S7_Templates := "SrcType := Int" } EQ_Contact(in1 := "BUFF".PROCESS, in2 := 73)
      I_Contact( "IEC_Timer_0_DB_90".Q )
   END_RUNG wire#w2
   RUNG wire#w1
      { S7_Templates := "SrcType := Int" } EQ_Contact(in1 := "BUFF".PROCESS, in2 := 60)
      I_Contact( "IEC_Timer_0_DB_94".Q )
   END_RUNG wire#w2
   RUNG wire#w1
      { S7_Templates := "SrcType := Int" } EQ_Contact(in1 := "BUFF".PROCESS, in2 := 80)
      I_Contact( "IEC_Timer_0_DB_88".Q )
   END_RUNG wire#w2
   RUNG wire#w1
      { S7_Templates := "SrcType := Int" } EQ_Contact(in1 := "BUFF".PROCESS, in2 := 152)
      { S7_Templates := "SrcType := Int" } NE_Contact(in1 := "AUXILIARY"."STD VCC HOLD", in2 := 0)
      I_Contact( "IEC_Timer_0_DB_96".Q )
   END_RUNG wire#w2
   // the same network as SCL:
   IF "AlwaysTRUE" AND ((("BUFF".PROCESS = 93) AND NOT "IEC_Timer_0_DB_84".Q) OR (("BUFF".PROCESS = 493) AND NOT "IEC_Timer_0_DB_196".Q) OR (("BUFF".PROCESS = 53) AND NOT "IEC_Timer_0_DB_91".Q) OR (("BUFF".PROCESS = 73) AND NOT "IEC_Timer_0_DB_90".Q) OR (("BUFF".PROCESS = 60) AND NOT "IEC_Timer_0_DB_94".Q) OR (("BUFF".PROCESS = 80) AND NOT "IEC_Timer_0_DB_88".Q) OR (("BUFF".PROCESS = 152) AND ("AUXILIARY"."STD VCC HOLD" <> 0) AND NOT "IEC_Timer_0_DB_96".Q)) THEN
       "REVAMP".CONVEYOR := ' HOLD END';
   END_IF;
END_REGION

REGION Network 15
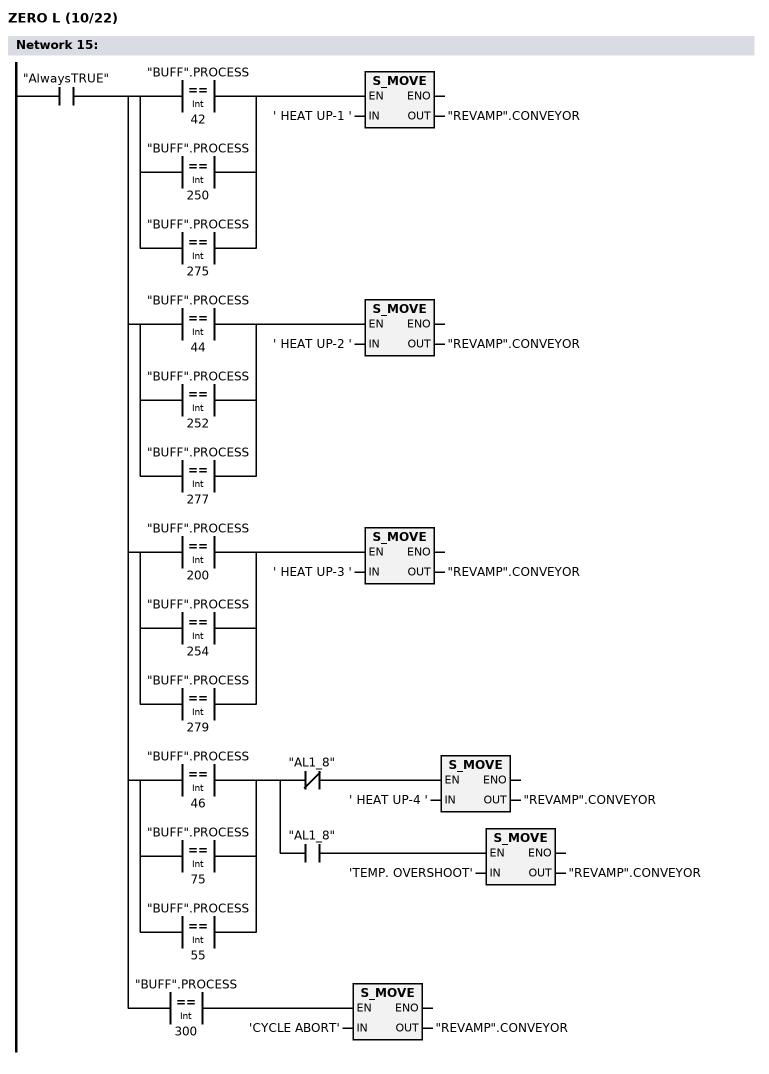
   RUNG wire#powerrail
      Contact( "AlwaysTRUE" )
      wire#w1
      { S7_Templates := "SrcType := Int" } EQ_Contact(in1 := "BUFF".PROCESS, in2 := 42)
      wire#w2
      S_Move(in := ' HEAT UP-1 ', out => "REVAMP".CONVEYOR)
   END_RUNG
   RUNG wire#w1
      { S7_Templates := "SrcType := Int" } EQ_Contact(in1 := "BUFF".PROCESS, in2 := 250)
   END_RUNG wire#w2
   RUNG wire#w1
      { S7_Templates := "SrcType := Int" } EQ_Contact(in1 := "BUFF".PROCESS, in2 := 275)
   END_RUNG wire#w2
   RUNG wire#w1
      { S7_Templates := "SrcType := Int" } EQ_Contact(in1 := "BUFF".PROCESS, in2 := 44)
      wire#w3
      S_Move(in := ' HEAT UP-2 ', out => "REVAMP".CONVEYOR)
   END_RUNG
   RUNG wire#w1
      { S7_Templates := "SrcType := Int" } EQ_Contact(in1 := "BUFF".PROCESS, in2 := 252)
   END_RUNG wire#w3
   RUNG wire#w1
      { S7_Templates := "SrcType := Int" } EQ_Contact(in1 := "BUFF".PROCESS, in2 := 277)
   END_RUNG wire#w3
   RUNG wire#w1
      { S7_Templates := "SrcType := Int" } EQ_Contact(in1 := "BUFF".PROCESS, in2 := 200)
      wire#w4
      S_Move(in := ' HEAT UP-3 ', out => "REVAMP".CONVEYOR)
   END_RUNG
   RUNG wire#w1
      { S7_Templates := "SrcType := Int" } EQ_Contact(in1 := "BUFF".PROCESS, in2 := 254)
   END_RUNG wire#w4
   RUNG wire#w1
      { S7_Templates := "SrcType := Int" } EQ_Contact(in1 := "BUFF".PROCESS, in2 := 279)
   END_RUNG wire#w4
   RUNG wire#w1
      { S7_Templates := "SrcType := Int" } EQ_Contact(in1 := "BUFF".PROCESS, in2 := 46)
      wire#w5
      I_Contact( "AL1_8" )
      S_Move(in := ' HEAT UP-4 ', out => "REVAMP".CONVEYOR)
   END_RUNG
   RUNG wire#w1
      { S7_Templates := "SrcType := Int" } EQ_Contact(in1 := "BUFF".PROCESS, in2 := 75)
   END_RUNG wire#w5
   RUNG wire#w1
      { S7_Templates := "SrcType := Int" } EQ_Contact(in1 := "BUFF".PROCESS, in2 := 55)
   END_RUNG wire#w5
   RUNG wire#w5
      Contact( "AL1_8" )
      S_Move(in := 'TEMP. OVERSHOOT', out => "REVAMP".CONVEYOR)
   END_RUNG
   RUNG wire#w1
      { S7_Templates := "SrcType := Int" } EQ_Contact(in1 := "BUFF".PROCESS, in2 := 300)
      S_Move(in := 'CYCLE ABORT', out => "REVAMP".CONVEYOR)
   END_RUNG
   // the same network as SCL:
   IF "AlwaysTRUE" AND (("BUFF".PROCESS = 42) OR ("BUFF".PROCESS = 250) OR ("BUFF".PROCESS = 275)) THEN
       "REVAMP".CONVEYOR := ' HEAT UP-1 ';
   END_IF;
   IF "AlwaysTRUE" AND (("BUFF".PROCESS = 44) OR ("BUFF".PROCESS = 252) OR ("BUFF".PROCESS = 277)) THEN
       "REVAMP".CONVEYOR := ' HEAT UP-2 ';
   END_IF;
   IF "AlwaysTRUE" AND (("BUFF".PROCESS = 200) OR ("BUFF".PROCESS = 254) OR ("BUFF".PROCESS = 279)) THEN
       "REVAMP".CONVEYOR := ' HEAT UP-3 ';
   END_IF;
   #_w1 := "AlwaysTRUE" AND (("BUFF".PROCESS = 46) OR ("BUFF".PROCESS = 75) OR ("BUFF".PROCESS = 55));
   IF #_w1 AND NOT "AL1_8" THEN "REVAMP".CONVEYOR := ' HEAT UP-4 '; END_IF;
   IF #_w1 AND "AL1_8" THEN "REVAMP".CONVEYOR := 'TEMP. OVERSHOOT'; END_IF;
   IF "AlwaysTRUE" AND ("BUFF".PROCESS = 300) THEN "REVAMP".CONVEYOR := 'CYCLE ABORT'; END_IF;
END_REGION

REGION Network 16
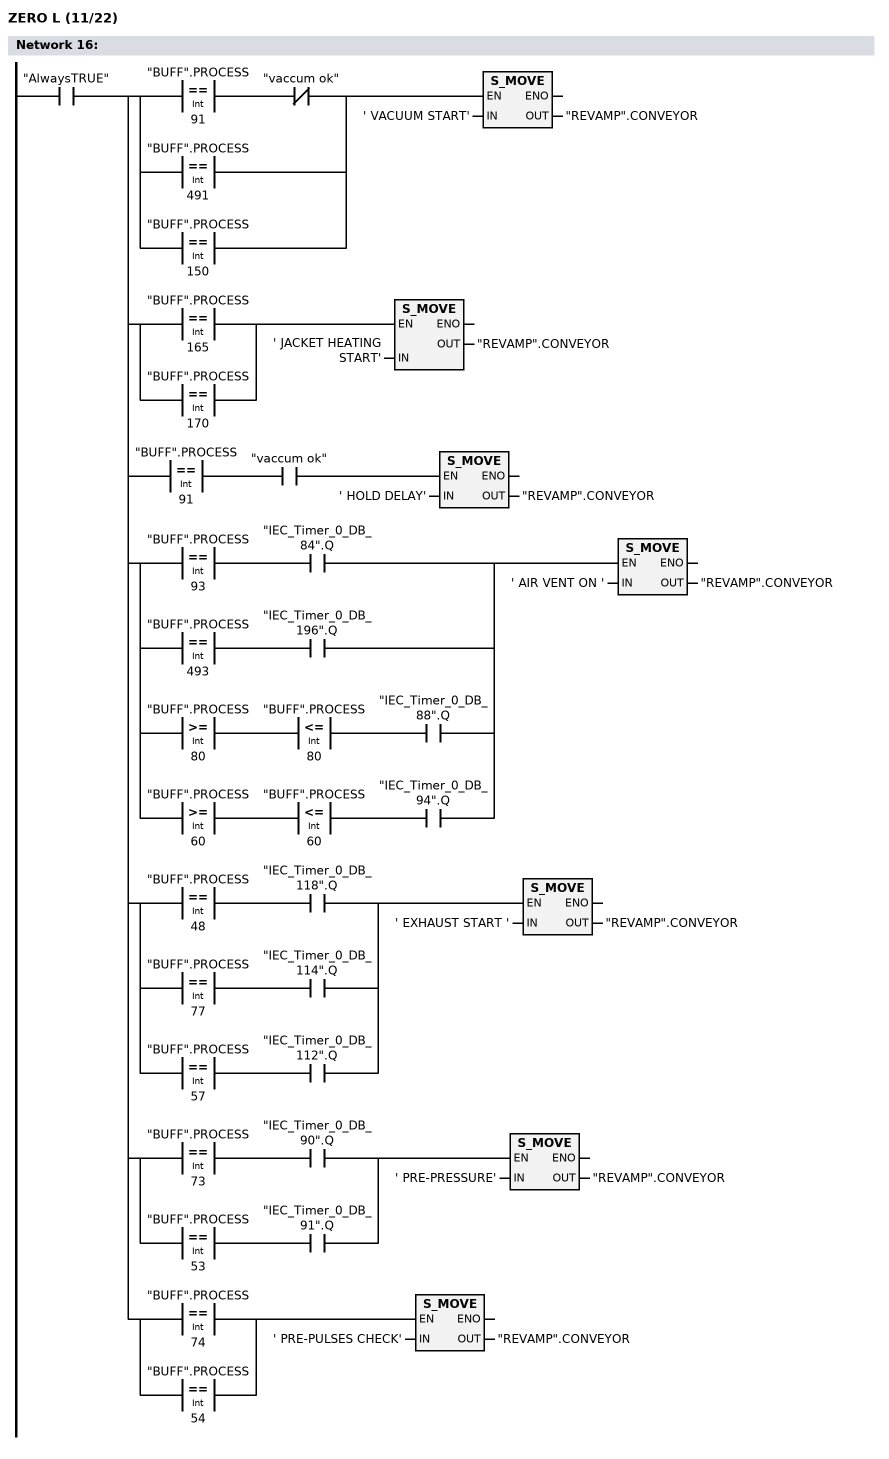
   RUNG wire#powerrail
      Contact( "AlwaysTRUE" )
      wire#w1
      { S7_Templates := "SrcType := Int" } EQ_Contact(in1 := "BUFF".PROCESS, in2 := 91)
      I_Contact( "vaccum ok" )
      wire#w2
      S_Move(in := ' VACUUM START', out => "REVAMP".CONVEYOR)
   END_RUNG
   RUNG wire#w1
      { S7_Templates := "SrcType := Int" } EQ_Contact(in1 := "BUFF".PROCESS, in2 := 491)
   END_RUNG wire#w2
   RUNG wire#w1
      { S7_Templates := "SrcType := Int" } EQ_Contact(in1 := "BUFF".PROCESS, in2 := 150)
   END_RUNG wire#w2
   RUNG wire#w1
      { S7_Templates := "SrcType := Int" } EQ_Contact(in1 := "BUFF".PROCESS, in2 := 165)
      wire#w3
      S_Move(in := ' JACKET HEATING START', out => "REVAMP".CONVEYOR)
   END_RUNG
   RUNG wire#w1
      { S7_Templates := "SrcType := Int" } EQ_Contact(in1 := "BUFF".PROCESS, in2 := 170)
   END_RUNG wire#w3
   RUNG wire#w1
      { S7_Templates := "SrcType := Int" } EQ_Contact(in1 := "BUFF".PROCESS, in2 := 91)
      Contact( "vaccum ok" )
      S_Move(in := ' HOLD DELAY', out => "REVAMP".CONVEYOR)
   END_RUNG
   RUNG wire#w1
      { S7_Templates := "SrcType := Int" } EQ_Contact(in1 := "BUFF".PROCESS, in2 := 93)
      Contact( "IEC_Timer_0_DB_84".Q )
      wire#w4
      S_Move(in := ' AIR VENT ON ', out => "REVAMP".CONVEYOR)
   END_RUNG
   RUNG wire#w1
      { S7_Templates := "SrcType := Int" } EQ_Contact(in1 := "BUFF".PROCESS, in2 := 493)
      Contact( "IEC_Timer_0_DB_196".Q )
   END_RUNG wire#w4
   RUNG wire#w1
      { S7_Templates := "SrcType := Int" } GE_Contact(in1 := "BUFF".PROCESS, in2 := 80)
      { S7_Templates := "SrcType := Int" } LE_Contact(in1 := "BUFF".PROCESS, in2 := 80)
      Contact( "IEC_Timer_0_DB_88".Q )
   END_RUNG wire#w4
   RUNG wire#w1
      { S7_Templates := "SrcType := Int" } GE_Contact(in1 := "BUFF".PROCESS, in2 := 60)
      { S7_Templates := "SrcType := Int" } LE_Contact(in1 := "BUFF".PROCESS, in2 := 60)
      Contact( "IEC_Timer_0_DB_94".Q )
   END_RUNG wire#w4
   RUNG wire#w1
      { S7_Templates := "SrcType := Int" } EQ_Contact(in1 := "BUFF".PROCESS, in2 := 48)
      Contact( "IEC_Timer_0_DB_118".Q )
      wire#w5
      S_Move(in := ' EXHAUST START ', out => "REVAMP".CONVEYOR)
   END_RUNG
   RUNG wire#w1
      { S7_Templates := "SrcType := Int" } EQ_Contact(in1 := "BUFF".PROCESS, in2 := 77)
      Contact( "IEC_Timer_0_DB_114".Q )
   END_RUNG wire#w5
   RUNG wire#w1
      { S7_Templates := "SrcType := Int" } EQ_Contact(in1 := "BUFF".PROCESS, in2 := 57)
      Contact( "IEC_Timer_0_DB_112".Q )
   END_RUNG wire#w5
   RUNG wire#w1
      { S7_Templates := "SrcType := Int" } EQ_Contact(in1 := "BUFF".PROCESS, in2 := 73)
      Contact( "IEC_Timer_0_DB_90".Q )
      wire#w6
      S_Move(in := ' PRE-PRESSURE', out => "REVAMP".CONVEYOR)
   END_RUNG
   RUNG wire#w1
      { S7_Templates := "SrcType := Int" } EQ_Contact(in1 := "BUFF".PROCESS, in2 := 53)
      Contact( "IEC_Timer_0_DB_91".Q )
   END_RUNG wire#w6
   RUNG wire#w1
      { S7_Templates := "SrcType := Int" } EQ_Contact(in1 := "BUFF".PROCESS, in2 := 74)
      wire#w7
      S_Move(in := ' PRE-PULSES CHECK', out => "REVAMP".CONVEYOR)
   END_RUNG
   RUNG wire#w1
      { S7_Templates := "SrcType := Int" } EQ_Contact(in1 := "BUFF".PROCESS, in2 := 54)
   END_RUNG wire#w7
   // the same network as SCL:
   IF "AlwaysTRUE" AND ((("BUFF".PROCESS = 91) AND NOT "vaccum ok") OR ("BUFF".PROCESS = 491) OR ("BUFF".PROCESS = 150)) THEN
       "REVAMP".CONVEYOR := ' VACUUM START';
   END_IF;
   IF "AlwaysTRUE" AND (("BUFF".PROCESS = 165) OR ("BUFF".PROCESS = 170)) THEN
       "REVAMP".CONVEYOR := ' JACKET HEATING START';
   END_IF;
   IF "AlwaysTRUE" AND ("BUFF".PROCESS = 91) AND "vaccum ok" THEN "REVAMP".CONVEYOR := ' HOLD DELAY'; END_IF;
   IF "AlwaysTRUE" AND ((("BUFF".PROCESS = 93) AND "IEC_Timer_0_DB_84".Q) OR (("BUFF".PROCESS = 493) AND "IEC_Timer_0_DB_196".Q) OR (("BUFF".PROCESS >= 80) AND ("BUFF".PROCESS <= 80) AND "IEC_Timer_0_DB_88".Q) OR (("BUFF".PROCESS >= 60) AND ("BUFF".PROCESS <= 60) AND "IEC_Timer_0_DB_94".Q)) THEN
       "REVAMP".CONVEYOR := ' AIR VENT ON ';
   END_IF;
   IF "AlwaysTRUE" AND ((("BUFF".PROCESS = 48) AND "IEC_Timer_0_DB_118".Q) OR (("BUFF".PROCESS = 77) AND "IEC_Timer_0_DB_114".Q) OR (("BUFF".PROCESS = 57) AND "IEC_Timer_0_DB_112".Q)) THEN
       "REVAMP".CONVEYOR := ' EXHAUST START ';
   END_IF;
   IF "AlwaysTRUE" AND ((("BUFF".PROCESS = 73) AND "IEC_Timer_0_DB_90".Q) OR (("BUFF".PROCESS = 53) AND "IEC_Timer_0_DB_91".Q)) THEN
       "REVAMP".CONVEYOR := ' PRE-PRESSURE';
   END_IF;
   IF "AlwaysTRUE" AND (("BUFF".PROCESS = 74) OR ("BUFF".PROCESS = 54)) THEN
       "REVAMP".CONVEYOR := ' PRE-PULSES CHECK';
   END_IF;
END_REGION

REGION Network 17
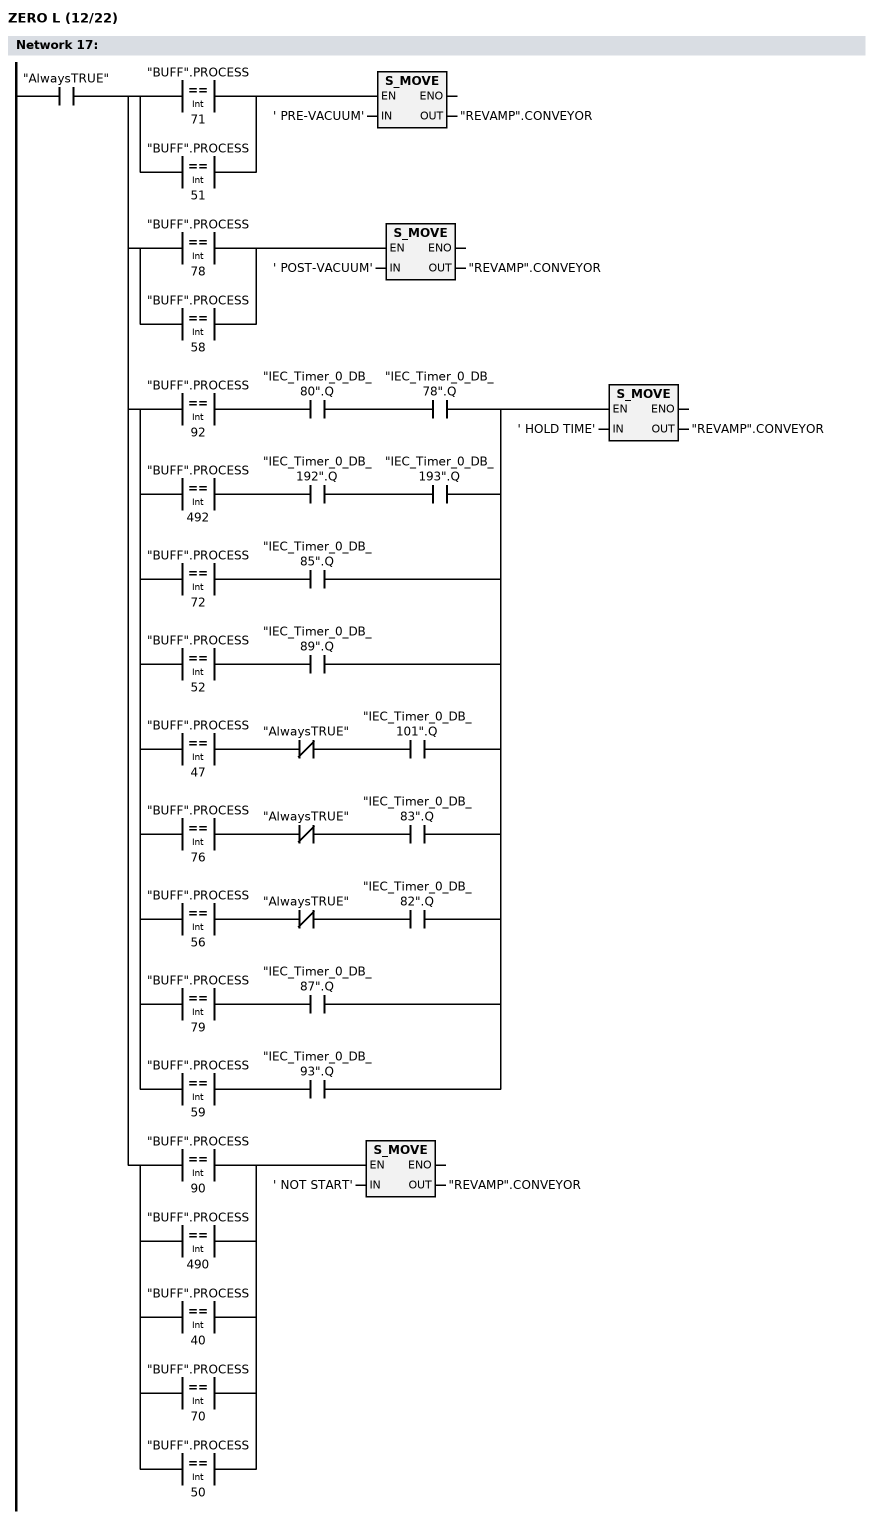
   RUNG wire#powerrail
      Contact( "AlwaysTRUE" )
      wire#w1
      { S7_Templates := "SrcType := Int" } EQ_Contact(in1 := "BUFF".PROCESS, in2 := 71)
      wire#w2
      S_Move(in := ' PRE-VACUUM', out => "REVAMP".CONVEYOR)
   END_RUNG
   RUNG wire#w1
      { S7_Templates := "SrcType := Int" } EQ_Contact(in1 := "BUFF".PROCESS, in2 := 51)
   END_RUNG wire#w2
   RUNG wire#w1
      { S7_Templates := "SrcType := Int" } EQ_Contact(in1 := "BUFF".PROCESS, in2 := 78)
      wire#w3
      S_Move(in := ' POST-VACUUM', out => "REVAMP".CONVEYOR)
   END_RUNG
   RUNG wire#w1
      { S7_Templates := "SrcType := Int" } EQ_Contact(in1 := "BUFF".PROCESS, in2 := 58)
   END_RUNG wire#w3
   RUNG wire#w1
      { S7_Templates := "SrcType := Int" } EQ_Contact(in1 := "BUFF".PROCESS, in2 := 92)
      Contact( "IEC_Timer_0_DB_80".Q )
      Contact( "IEC_Timer_0_DB_78".Q )
      wire#w4
      S_Move(in := ' HOLD TIME', out => "REVAMP".CONVEYOR)
   END_RUNG
   RUNG wire#w1
      { S7_Templates := "SrcType := Int" } EQ_Contact(in1 := "BUFF".PROCESS, in2 := 492)
      Contact( "IEC_Timer_0_DB_192".Q )
      Contact( "IEC_Timer_0_DB_193".Q )
   END_RUNG wire#w4
   RUNG wire#w1
      { S7_Templates := "SrcType := Int" } EQ_Contact(in1 := "BUFF".PROCESS, in2 := 72)
      Contact( "IEC_Timer_0_DB_85".Q )
   END_RUNG wire#w4
   RUNG wire#w1
      { S7_Templates := "SrcType := Int" } EQ_Contact(in1 := "BUFF".PROCESS, in2 := 52)
      Contact( "IEC_Timer_0_DB_89".Q )
   END_RUNG wire#w4
   RUNG wire#w1
      { S7_Templates := "SrcType := Int" } EQ_Contact(in1 := "BUFF".PROCESS, in2 := 47)
      I_Contact( "AlwaysTRUE" )
      Contact( "IEC_Timer_0_DB_101".Q )
   END_RUNG wire#w4
   RUNG wire#w1
      { S7_Templates := "SrcType := Int" } EQ_Contact(in1 := "BUFF".PROCESS, in2 := 76)
      I_Contact( "AlwaysTRUE" )
      Contact( "IEC_Timer_0_DB_83".Q )
   END_RUNG wire#w4
   RUNG wire#w1
      { S7_Templates := "SrcType := Int" } EQ_Contact(in1 := "BUFF".PROCESS, in2 := 56)
      I_Contact( "AlwaysTRUE" )
      Contact( "IEC_Timer_0_DB_82".Q )
   END_RUNG wire#w4
   RUNG wire#w1
      { S7_Templates := "SrcType := Int" } EQ_Contact(in1 := "BUFF".PROCESS, in2 := 79)
      Contact( "IEC_Timer_0_DB_87".Q )
   END_RUNG wire#w4
   RUNG wire#w1
      { S7_Templates := "SrcType := Int" } EQ_Contact(in1 := "BUFF".PROCESS, in2 := 59)
      Contact( "IEC_Timer_0_DB_93".Q )
   END_RUNG wire#w4
   RUNG wire#w1
      { S7_Templates := "SrcType := Int" } EQ_Contact(in1 := "BUFF".PROCESS, in2 := 90)
      wire#w5
      S_Move(in := ' NOT START', out => "REVAMP".CONVEYOR)
   END_RUNG
   RUNG wire#w1
      { S7_Templates := "SrcType := Int" } EQ_Contact(in1 := "BUFF".PROCESS, in2 := 490)
   END_RUNG wire#w5
   RUNG wire#w1
      { S7_Templates := "SrcType := Int" } EQ_Contact(in1 := "BUFF".PROCESS, in2 := 40)
   END_RUNG wire#w5
   RUNG wire#w1
      { S7_Templates := "SrcType := Int" } EQ_Contact(in1 := "BUFF".PROCESS, in2 := 70)
   END_RUNG wire#w5
   RUNG wire#w1
      { S7_Templates := "SrcType := Int" } EQ_Contact(in1 := "BUFF".PROCESS, in2 := 50)
   END_RUNG wire#w5
   // the same network as SCL:
   IF "AlwaysTRUE" AND (("BUFF".PROCESS = 71) OR ("BUFF".PROCESS = 51)) THEN
       "REVAMP".CONVEYOR := ' PRE-VACUUM';
   END_IF;
   IF "AlwaysTRUE" AND (("BUFF".PROCESS = 78) OR ("BUFF".PROCESS = 58)) THEN
       "REVAMP".CONVEYOR := ' POST-VACUUM';
   END_IF;
   IF "AlwaysTRUE" AND ((("BUFF".PROCESS = 92) AND "IEC_Timer_0_DB_80".Q AND "IEC_Timer_0_DB_78".Q) OR (("BUFF".PROCESS = 492) AND "IEC_Timer_0_DB_192".Q AND "IEC_Timer_0_DB_193".Q) OR (("BUFF".PROCESS = 72) AND "IEC_Timer_0_DB_85".Q) OR (("BUFF".PROCESS = 52) AND "IEC_Timer_0_DB_89".Q) OR (("BUFF".PROCESS = 47) AND NOT "AlwaysTRUE" AND "IEC_Timer_0_DB_101".Q) OR (("BUFF".PROCESS = 76) AND NOT "AlwaysTRUE" AND "IEC_Timer_0_DB_83".Q) OR (("BUFF".PROCESS = 56) AND NOT "AlwaysTRUE" AND "IEC_Timer_0_DB_82".Q) OR (("BUFF".PROCESS = 79) AND "IEC_Timer_0_DB_87".Q) OR (("BUFF".PROCESS = 59) AND "IEC_Timer_0_DB_93".Q)) THEN
       "REVAMP".CONVEYOR := ' HOLD TIME';
   END_IF;
   IF "AlwaysTRUE" AND (("BUFF".PROCESS = 90) OR ("BUFF".PROCESS = 490) OR ("BUFF".PROCESS = 40) OR ("BUFF".PROCESS = 70) OR ("BUFF".PROCESS = 50)) THEN
       "REVAMP".CONVEYOR := ' NOT START';
   END_IF;
END_REGION

REGION Network 18
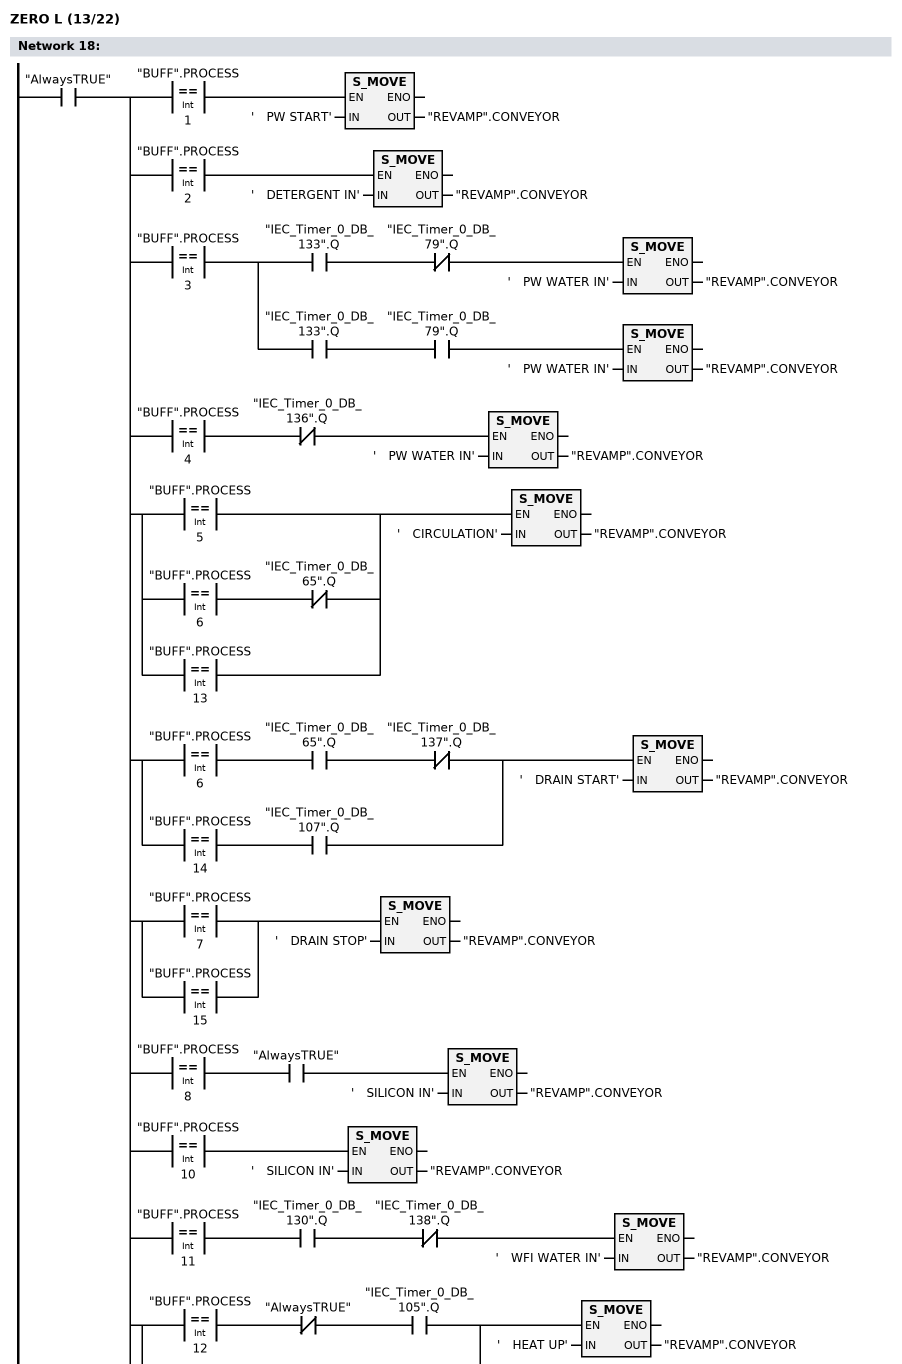
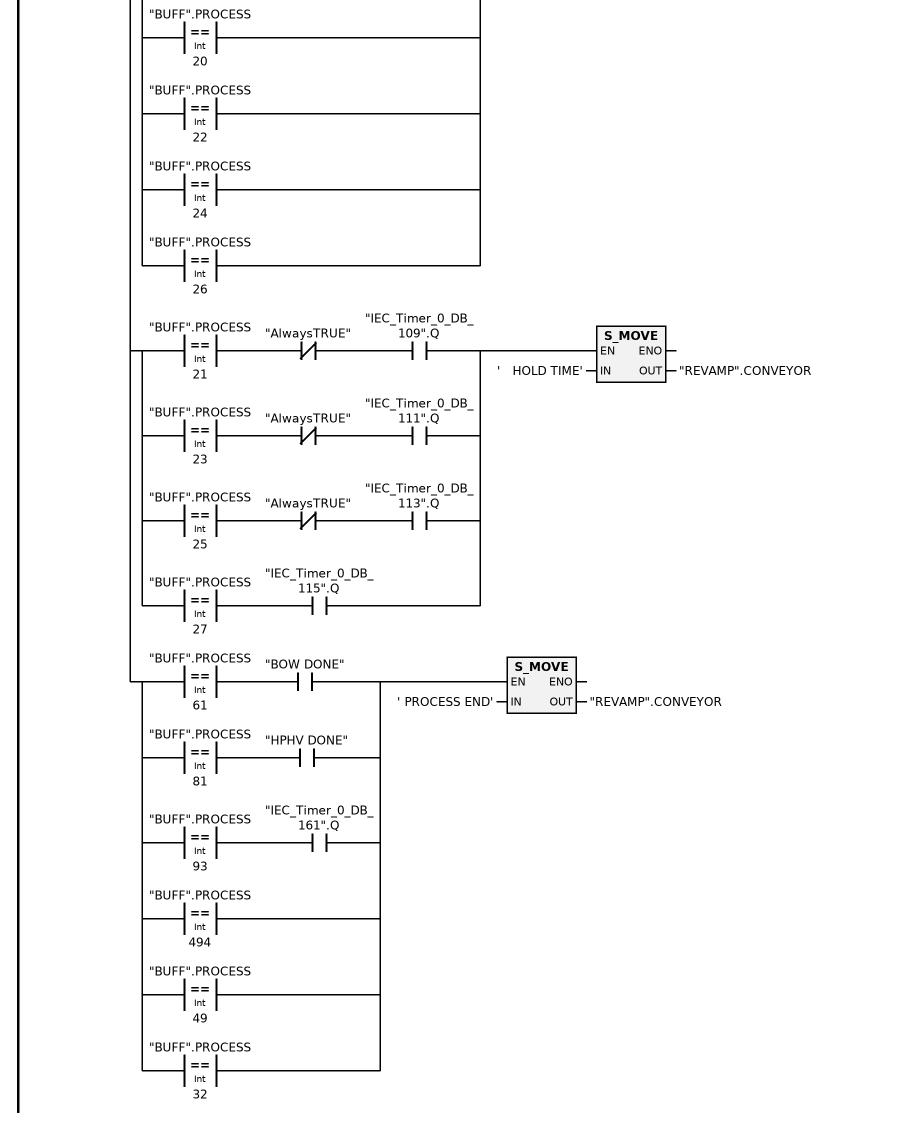
   RUNG wire#powerrail
      Contact( "AlwaysTRUE" )
      wire#w1
      { S7_Templates := "SrcType := Int" } EQ_Contact(in1 := "BUFF".PROCESS, in2 := 1)
      S_Move(in := '   PW START', out => "REVAMP".CONVEYOR)
   END_RUNG
   RUNG wire#w1
      { S7_Templates := "SrcType := Int" } EQ_Contact(in1 := "BUFF".PROCESS, in2 := 2)
      S_Move(in := '   DETERGENT IN', out => "REVAMP".CONVEYOR)
   END_RUNG
   RUNG wire#w1
      { S7_Templates := "SrcType := Int" } EQ_Contact(in1 := "BUFF".PROCESS, in2 := 3)
      wire#w2
      Contact( "IEC_Timer_0_DB_133".Q )
      I_Contact( "IEC_Timer_0_DB_79".Q )
      S_Move(in := '   PW WATER IN', out => "REVAMP".CONVEYOR)
   END_RUNG
   RUNG wire#w2
      Contact( "IEC_Timer_0_DB_133".Q )
      Contact( "IEC_Timer_0_DB_79".Q )
      S_Move(in := '   PW WATER IN', out => "REVAMP".CONVEYOR)
   END_RUNG
   RUNG wire#w1
      { S7_Templates := "SrcType := Int" } EQ_Contact(in1 := "BUFF".PROCESS, in2 := 4)
      I_Contact( "IEC_Timer_0_DB_136".Q )
      S_Move(in := '   PW WATER IN', out => "REVAMP".CONVEYOR)
   END_RUNG
   RUNG wire#w1
      { S7_Templates := "SrcType := Int" } EQ_Contact(in1 := "BUFF".PROCESS, in2 := 5)
      wire#w3
      S_Move(in := '   CIRCULATION', out => "REVAMP".CONVEYOR)
   END_RUNG
   RUNG wire#w1
      { S7_Templates := "SrcType := Int" } EQ_Contact(in1 := "BUFF".PROCESS, in2 := 6)
      I_Contact( "IEC_Timer_0_DB_65".Q )
   END_RUNG wire#w3
   RUNG wire#w1
      { S7_Templates := "SrcType := Int" } EQ_Contact(in1 := "BUFF".PROCESS, in2 := 13)
   END_RUNG wire#w3
   RUNG wire#w1
      { S7_Templates := "SrcType := Int" } EQ_Contact(in1 := "BUFF".PROCESS, in2 := 6)
      Contact( "IEC_Timer_0_DB_65".Q )
      I_Contact( "IEC_Timer_0_DB_137".Q )
      wire#w4
      S_Move(in := '   DRAIN START', out => "REVAMP".CONVEYOR)
   END_RUNG
   RUNG wire#w1
      { S7_Templates := "SrcType := Int" } EQ_Contact(in1 := "BUFF".PROCESS, in2 := 14)
      Contact( "IEC_Timer_0_DB_107".Q )
   END_RUNG wire#w4
   RUNG wire#w1
      { S7_Templates := "SrcType := Int" } EQ_Contact(in1 := "BUFF".PROCESS, in2 := 7)
      wire#w5
      S_Move(in := '   DRAIN STOP', out => "REVAMP".CONVEYOR)
   END_RUNG
   RUNG wire#w1
      { S7_Templates := "SrcType := Int" } EQ_Contact(in1 := "BUFF".PROCESS, in2 := 15)
   END_RUNG wire#w5
   RUNG wire#w1
      { S7_Templates := "SrcType := Int" } EQ_Contact(in1 := "BUFF".PROCESS, in2 := 8)
      Contact( "AlwaysTRUE" )
      S_Move(in := '   SILICON IN', out => "REVAMP".CONVEYOR)
   END_RUNG
   RUNG wire#w1
      { S7_Templates := "SrcType := Int" } EQ_Contact(in1 := "BUFF".PROCESS, in2 := 10)
      S_Move(in := '   SILICON IN', out => "REVAMP".CONVEYOR)
   END_RUNG
   RUNG wire#w1
      { S7_Templates := "SrcType := Int" } EQ_Contact(in1 := "BUFF".PROCESS, in2 := 11)
      Contact( "IEC_Timer_0_DB_130".Q )
      I_Contact( "IEC_Timer_0_DB_138".Q )
      S_Move(in := '   WFI WATER IN', out => "REVAMP".CONVEYOR)
   END_RUNG
   RUNG wire#w1
      { S7_Templates := "SrcType := Int" } EQ_Contact(in1 := "BUFF".PROCESS, in2 := 12)
      I_Contact( "AlwaysTRUE" )
      Contact( "IEC_Timer_0_DB_105".Q )
      wire#w6
      S_Move(in := '   HEAT UP', out => "REVAMP".CONVEYOR)
   END_RUNG
   RUNG wire#w1
      { S7_Templates := "SrcType := Int" } EQ_Contact(in1 := "BUFF".PROCESS, in2 := 20)
   END_RUNG wire#w6
   RUNG wire#w1
      { S7_Templates := "SrcType := Int" } EQ_Contact(in1 := "BUFF".PROCESS, in2 := 22)
   END_RUNG wire#w6
   RUNG wire#w1
      { S7_Templates := "SrcType := Int" } EQ_Contact(in1 := "BUFF".PROCESS, in2 := 24)
   END_RUNG wire#w6
   RUNG wire#w1
      { S7_Templates := "SrcType := Int" } EQ_Contact(in1 := "BUFF".PROCESS, in2 := 26)
   END_RUNG wire#w6
   RUNG wire#w1
      { S7_Templates := "SrcType := Int" } EQ_Contact(in1 := "BUFF".PROCESS, in2 := 21)
      I_Contact( "AlwaysTRUE" )
      Contact( "IEC_Timer_0_DB_109".Q )
      wire#w7
      S_Move(in := '   HOLD TIME', out => "REVAMP".CONVEYOR)
   END_RUNG
   RUNG wire#w1
      { S7_Templates := "SrcType := Int" } EQ_Contact(in1 := "BUFF".PROCESS, in2 := 23)
      I_Contact( "AlwaysTRUE" )
      Contact( "IEC_Timer_0_DB_111".Q )
   END_RUNG wire#w7
   RUNG wire#w1
      { S7_Templates := "SrcType := Int" } EQ_Contact(in1 := "BUFF".PROCESS, in2 := 25)
      I_Contact( "AlwaysTRUE" )
      Contact( "IEC_Timer_0_DB_113".Q )
   END_RUNG wire#w7
   RUNG wire#w1
      { S7_Templates := "SrcType := Int" } EQ_Contact(in1 := "BUFF".PROCESS, in2 := 27)
      Contact( "IEC_Timer_0_DB_115".Q )
   END_RUNG wire#w7
   RUNG wire#w1
      { S7_Templates := "SrcType := Int" } EQ_Contact(in1 := "BUFF".PROCESS, in2 := 61)
      Contact( "BOW DONE" )
      wire#w8
      S_Move(in := ' PROCESS END', out => "REVAMP".CONVEYOR)
   END_RUNG
   RUNG wire#w1
      { S7_Templates := "SrcType := Int" } EQ_Contact(in1 := "BUFF".PROCESS, in2 := 81)
      Contact( "HPHV DONE" )
   END_RUNG wire#w8
   RUNG wire#w1
      { S7_Templates := "SrcType := Int" } EQ_Contact(in1 := "BUFF".PROCESS, in2 := 93)
      Contact( "IEC_Timer_0_DB_161".Q )
   END_RUNG wire#w8
   RUNG wire#w1
      { S7_Templates := "SrcType := Int" } EQ_Contact(in1 := "BUFF".PROCESS, in2 := 494)
   END_RUNG wire#w8
   RUNG wire#w1
      { S7_Templates := "SrcType := Int" } EQ_Contact(in1 := "BUFF".PROCESS, in2 := 49)
   END_RUNG wire#w8
   RUNG wire#w1
      { S7_Templates := "SrcType := Int" } EQ_Contact(in1 := "BUFF".PROCESS, in2 := 32)
   END_RUNG wire#w8
   // the same network as SCL:
   IF "AlwaysTRUE" AND ("BUFF".PROCESS = 1) THEN "REVAMP".CONVEYOR := '   PW START'; END_IF;
   IF "AlwaysTRUE" AND ("BUFF".PROCESS = 2) THEN "REVAMP".CONVEYOR := '   DETERGENT IN'; END_IF;
   #_w1 := "AlwaysTRUE" AND ("BUFF".PROCESS = 3);
   IF #_w1 AND "IEC_Timer_0_DB_133".Q AND NOT "IEC_Timer_0_DB_79".Q THEN
       "REVAMP".CONVEYOR := '   PW WATER IN';
   END_IF;
   IF #_w1 AND "IEC_Timer_0_DB_133".Q AND "IEC_Timer_0_DB_79".Q THEN
       "REVAMP".CONVEYOR := '   PW WATER IN';
   END_IF;
   IF "AlwaysTRUE" AND ("BUFF".PROCESS = 4) AND NOT "IEC_Timer_0_DB_136".Q THEN
       "REVAMP".CONVEYOR := '   PW WATER IN';
   END_IF;
   IF "AlwaysTRUE" AND (("BUFF".PROCESS = 5) OR (("BUFF".PROCESS = 6) AND NOT "IEC_Timer_0_DB_65".Q) OR ("BUFF".PROCESS = 13)) THEN
       "REVAMP".CONVEYOR := '   CIRCULATION';
   END_IF;
   IF "AlwaysTRUE" AND ((("BUFF".PROCESS = 6) AND "IEC_Timer_0_DB_65".Q AND NOT "IEC_Timer_0_DB_137".Q) OR (("BUFF".PROCESS = 14) AND "IEC_Timer_0_DB_107".Q)) THEN
       "REVAMP".CONVEYOR := '   DRAIN START';
   END_IF;
   IF "AlwaysTRUE" AND (("BUFF".PROCESS = 7) OR ("BUFF".PROCESS = 15)) THEN
       "REVAMP".CONVEYOR := '   DRAIN STOP';
   END_IF;
   IF "AlwaysTRUE" AND ("BUFF".PROCESS = 8) AND "AlwaysTRUE" THEN
       "REVAMP".CONVEYOR := '   SILICON IN';
   END_IF;
   IF "AlwaysTRUE" AND ("BUFF".PROCESS = 10) THEN "REVAMP".CONVEYOR := '   SILICON IN'; END_IF;
   IF "AlwaysTRUE" AND ("BUFF".PROCESS = 11) AND "IEC_Timer_0_DB_130".Q AND NOT "IEC_Timer_0_DB_138".Q THEN
       "REVAMP".CONVEYOR := '   WFI WATER IN';
   END_IF;
   IF "AlwaysTRUE" AND ((("BUFF".PROCESS = 12) AND NOT "AlwaysTRUE" AND "IEC_Timer_0_DB_105".Q) OR ("BUFF".PROCESS = 20) OR ("BUFF".PROCESS = 22) OR ("BUFF".PROCESS = 24) OR ("BUFF".PROCESS = 26)) THEN
       "REVAMP".CONVEYOR := '   HEAT UP';
   END_IF;
   IF "AlwaysTRUE" AND ((("BUFF".PROCESS = 21) AND NOT "AlwaysTRUE" AND "IEC_Timer_0_DB_109".Q) OR (("BUFF".PROCESS = 23) AND NOT "AlwaysTRUE" AND "IEC_Timer_0_DB_111".Q) OR (("BUFF".PROCESS = 25) AND NOT "AlwaysTRUE" AND "IEC_Timer_0_DB_113".Q) OR (("BUFF".PROCESS = 27) AND "IEC_Timer_0_DB_115".Q)) THEN
       "REVAMP".CONVEYOR := '   HOLD TIME';
   END_IF;
   IF "AlwaysTRUE" AND ((("BUFF".PROCESS = 61) AND "BOW DONE") OR (("BUFF".PROCESS = 81) AND "HPHV DONE") OR (("BUFF".PROCESS = 93) AND "IEC_Timer_0_DB_161".Q) OR ("BUFF".PROCESS = 494) OR ("BUFF".PROCESS = 49) OR ("BUFF".PROCESS = 32)) THEN
       "REVAMP".CONVEYOR := ' PROCESS END';
   END_IF;
END_REGION

REGION Network 19
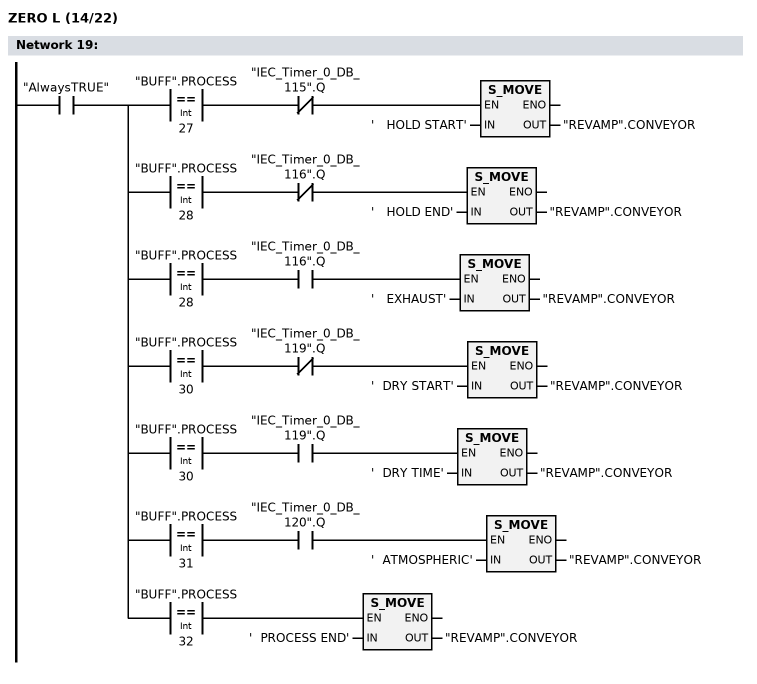
   RUNG wire#powerrail
      Contact( "AlwaysTRUE" )
      wire#w1
      { S7_Templates := "SrcType := Int" } EQ_Contact(in1 := "BUFF".PROCESS, in2 := 27)
      I_Contact( "IEC_Timer_0_DB_115".Q )
      S_Move(in := '   HOLD START', out => "REVAMP".CONVEYOR)
   END_RUNG
   RUNG wire#w1
      { S7_Templates := "SrcType := Int" } EQ_Contact(in1 := "BUFF".PROCESS, in2 := 28)
      I_Contact( "IEC_Timer_0_DB_116".Q )
      S_Move(in := '   HOLD END', out => "REVAMP".CONVEYOR)
   END_RUNG
   RUNG wire#w1
      { S7_Templates := "SrcType := Int" } EQ_Contact(in1 := "BUFF".PROCESS, in2 := 28)
      Contact( "IEC_Timer_0_DB_116".Q )
      S_Move(in := '   EXHAUST', out => "REVAMP".CONVEYOR)
   END_RUNG
   RUNG wire#w1
      { S7_Templates := "SrcType := Int" } EQ_Contact(in1 := "BUFF".PROCESS, in2 := 30)
      I_Contact( "IEC_Timer_0_DB_119".Q )
      S_Move(in := '  DRY START', out => "REVAMP".CONVEYOR)
   END_RUNG
   RUNG wire#w1
      { S7_Templates := "SrcType := Int" } EQ_Contact(in1 := "BUFF".PROCESS, in2 := 30)
      Contact( "IEC_Timer_0_DB_119".Q )
      S_Move(in := '  DRY TIME', out => "REVAMP".CONVEYOR)
   END_RUNG
   RUNG wire#w1
      { S7_Templates := "SrcType := Int" } EQ_Contact(in1 := "BUFF".PROCESS, in2 := 31)
      Contact( "IEC_Timer_0_DB_120".Q )
      S_Move(in := '  ATMOSPHERIC', out => "REVAMP".CONVEYOR)
   END_RUNG
   RUNG wire#w1
      { S7_Templates := "SrcType := Int" } EQ_Contact(in1 := "BUFF".PROCESS, in2 := 32)
      S_Move(in := '  PROCESS END', out => "REVAMP".CONVEYOR)
   END_RUNG
   // the same network as SCL:
   IF "AlwaysTRUE" AND ("BUFF".PROCESS = 27) AND NOT "IEC_Timer_0_DB_115".Q THEN
       "REVAMP".CONVEYOR := '   HOLD START';
   END_IF;
   IF "AlwaysTRUE" AND ("BUFF".PROCESS = 28) AND NOT "IEC_Timer_0_DB_116".Q THEN
       "REVAMP".CONVEYOR := '   HOLD END';
   END_IF;
   IF "AlwaysTRUE" AND ("BUFF".PROCESS = 28) AND "IEC_Timer_0_DB_116".Q THEN
       "REVAMP".CONVEYOR := '   EXHAUST';
   END_IF;
   IF "AlwaysTRUE" AND ("BUFF".PROCESS = 30) AND NOT "IEC_Timer_0_DB_119".Q THEN
       "REVAMP".CONVEYOR := '  DRY START';
   END_IF;
   IF "AlwaysTRUE" AND ("BUFF".PROCESS = 30) AND "IEC_Timer_0_DB_119".Q THEN
       "REVAMP".CONVEYOR := '  DRY TIME';
   END_IF;
   IF "AlwaysTRUE" AND ("BUFF".PROCESS = 31) AND "IEC_Timer_0_DB_120".Q THEN
       "REVAMP".CONVEYOR := '  ATMOSPHERIC';
   END_IF;
   IF "AlwaysTRUE" AND ("BUFF".PROCESS = 32) THEN "REVAMP".CONVEYOR := '  PROCESS END'; END_IF;
END_REGION

REGION Network 20
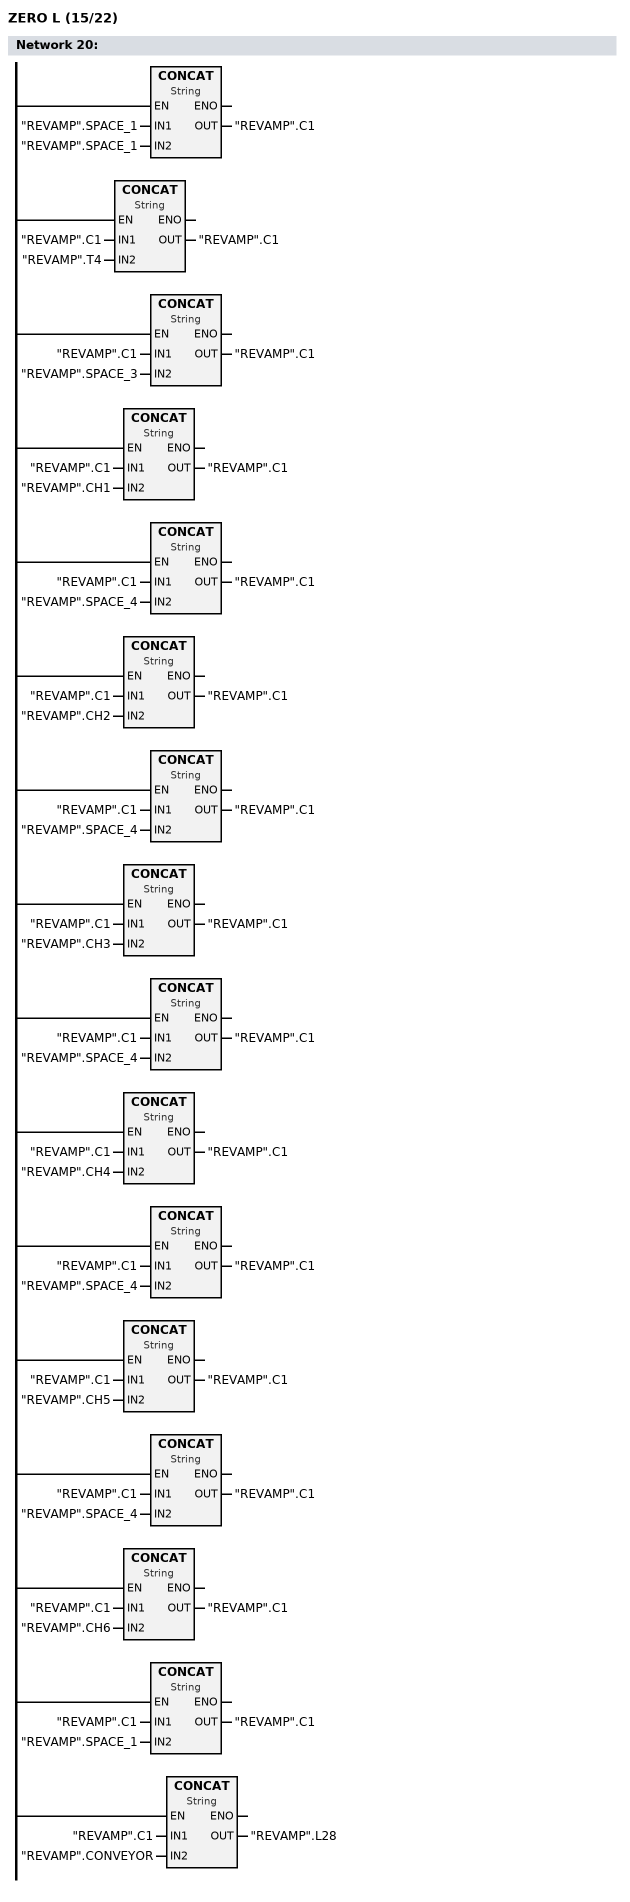
   RUNG wire#powerrail
      { S7_Templates := "[card := 2, str_type := String]" } CONCAT(IN1 := "REVAMP".SPACE_1, IN2 := "REVAMP".SPACE_1, OUT => "REVAMP".C1)
   END_RUNG
   RUNG wire#powerrail
      { S7_Templates := "[card := 2, str_type := String]" } CONCAT(IN1 := "REVAMP".C1, IN2 := "REVAMP".T4, OUT => "REVAMP".C1)
   END_RUNG
   RUNG wire#powerrail
      { S7_Templates := "[card := 2, str_type := String]" } CONCAT(IN1 := "REVAMP".C1, IN2 := "REVAMP".SPACE_3, OUT => "REVAMP".C1)
   END_RUNG
   RUNG wire#powerrail
      { S7_Templates := "[card := 2, str_type := String]" } CONCAT(IN1 := "REVAMP".C1, IN2 := "REVAMP".CH1, OUT => "REVAMP".C1)
   END_RUNG
   RUNG wire#powerrail
      { S7_Templates := "[card := 2, str_type := String]" } CONCAT(IN1 := "REVAMP".C1, IN2 := "REVAMP".SPACE_4, OUT => "REVAMP".C1)
   END_RUNG
   RUNG wire#powerrail
      { S7_Templates := "[card := 2, str_type := String]" } CONCAT(IN1 := "REVAMP".C1, IN2 := "REVAMP".CH2, OUT => "REVAMP".C1)
   END_RUNG
   RUNG wire#powerrail
      { S7_Templates := "[card := 2, str_type := String]" } CONCAT(IN1 := "REVAMP".C1, IN2 := "REVAMP".SPACE_4, OUT => "REVAMP".C1)
   END_RUNG
   RUNG wire#powerrail
      { S7_Templates := "[card := 2, str_type := String]" } CONCAT(IN1 := "REVAMP".C1, IN2 := "REVAMP".CH3, OUT => "REVAMP".C1)
   END_RUNG
   RUNG wire#powerrail
      { S7_Templates := "[card := 2, str_type := String]" } CONCAT(IN1 := "REVAMP".C1, IN2 := "REVAMP".SPACE_4, OUT => "REVAMP".C1)
   END_RUNG
   RUNG wire#powerrail
      { S7_Templates := "[card := 2, str_type := String]" } CONCAT(IN1 := "REVAMP".C1, IN2 := "REVAMP".CH4, OUT => "REVAMP".C1)
   END_RUNG
   RUNG wire#powerrail
      { S7_Templates := "[card := 2, str_type := String]" } CONCAT(IN1 := "REVAMP".C1, IN2 := "REVAMP".SPACE_4, OUT => "REVAMP".C1)
   END_RUNG
   RUNG wire#powerrail
      { S7_Templates := "[card := 2, str_type := String]" } CONCAT(IN1 := "REVAMP".C1, IN2 := "REVAMP".CH5, OUT => "REVAMP".C1)
   END_RUNG
   RUNG wire#powerrail
      { S7_Templates := "[card := 2, str_type := String]" } CONCAT(IN1 := "REVAMP".C1, IN2 := "REVAMP".SPACE_4, OUT => "REVAMP".C1)
   END_RUNG
   RUNG wire#powerrail
      { S7_Templates := "[card := 2, str_type := String]" } CONCAT(IN1 := "REVAMP".C1, IN2 := "REVAMP".CH6, OUT => "REVAMP".C1)
   END_RUNG
   RUNG wire#powerrail
      { S7_Templates := "[card := 2, str_type := String]" } CONCAT(IN1 := "REVAMP".C1, IN2 := "REVAMP".SPACE_1, OUT => "REVAMP".C1)
   END_RUNG
   RUNG wire#powerrail
      { S7_Templates := "[card := 2, str_type := String]" } CONCAT(IN1 := "REVAMP".C1, IN2 := "REVAMP".CONVEYOR, OUT => "REVAMP".L28)
   END_RUNG
   // the same network as SCL:
   CONCAT(IN1 := "REVAMP".SPACE_1, IN2 := "REVAMP".SPACE_1, OUT => "REVAMP".C1);
   CONCAT(IN1 := "REVAMP".C1, IN2 := "REVAMP".T4, OUT => "REVAMP".C1);
   CONCAT(IN1 := "REVAMP".C1, IN2 := "REVAMP".SPACE_3, OUT => "REVAMP".C1);
   CONCAT(IN1 := "REVAMP".C1, IN2 := "REVAMP".CH1, OUT => "REVAMP".C1);
   CONCAT(IN1 := "REVAMP".C1, IN2 := "REVAMP".SPACE_4, OUT => "REVAMP".C1);
   CONCAT(IN1 := "REVAMP".C1, IN2 := "REVAMP".CH2, OUT => "REVAMP".C1);
   CONCAT(IN1 := "REVAMP".C1, IN2 := "REVAMP".SPACE_4, OUT => "REVAMP".C1);
   CONCAT(IN1 := "REVAMP".C1, IN2 := "REVAMP".CH3, OUT => "REVAMP".C1);
   CONCAT(IN1 := "REVAMP".C1, IN2 := "REVAMP".SPACE_4, OUT => "REVAMP".C1);
   CONCAT(IN1 := "REVAMP".C1, IN2 := "REVAMP".CH4, OUT => "REVAMP".C1);
   CONCAT(IN1 := "REVAMP".C1, IN2 := "REVAMP".SPACE_4, OUT => "REVAMP".C1);
   CONCAT(IN1 := "REVAMP".C1, IN2 := "REVAMP".CH5, OUT => "REVAMP".C1);
   CONCAT(IN1 := "REVAMP".C1, IN2 := "REVAMP".SPACE_4, OUT => "REVAMP".C1);
   CONCAT(IN1 := "REVAMP".C1, IN2 := "REVAMP".CH6, OUT => "REVAMP".C1);
   CONCAT(IN1 := "REVAMP".C1, IN2 := "REVAMP".SPACE_1, OUT => "REVAMP".C1);
   CONCAT(IN1 := "REVAMP".C1, IN2 := "REVAMP".CONVEYOR, OUT => "REVAMP".L28);
END_REGION

REGION Network 21
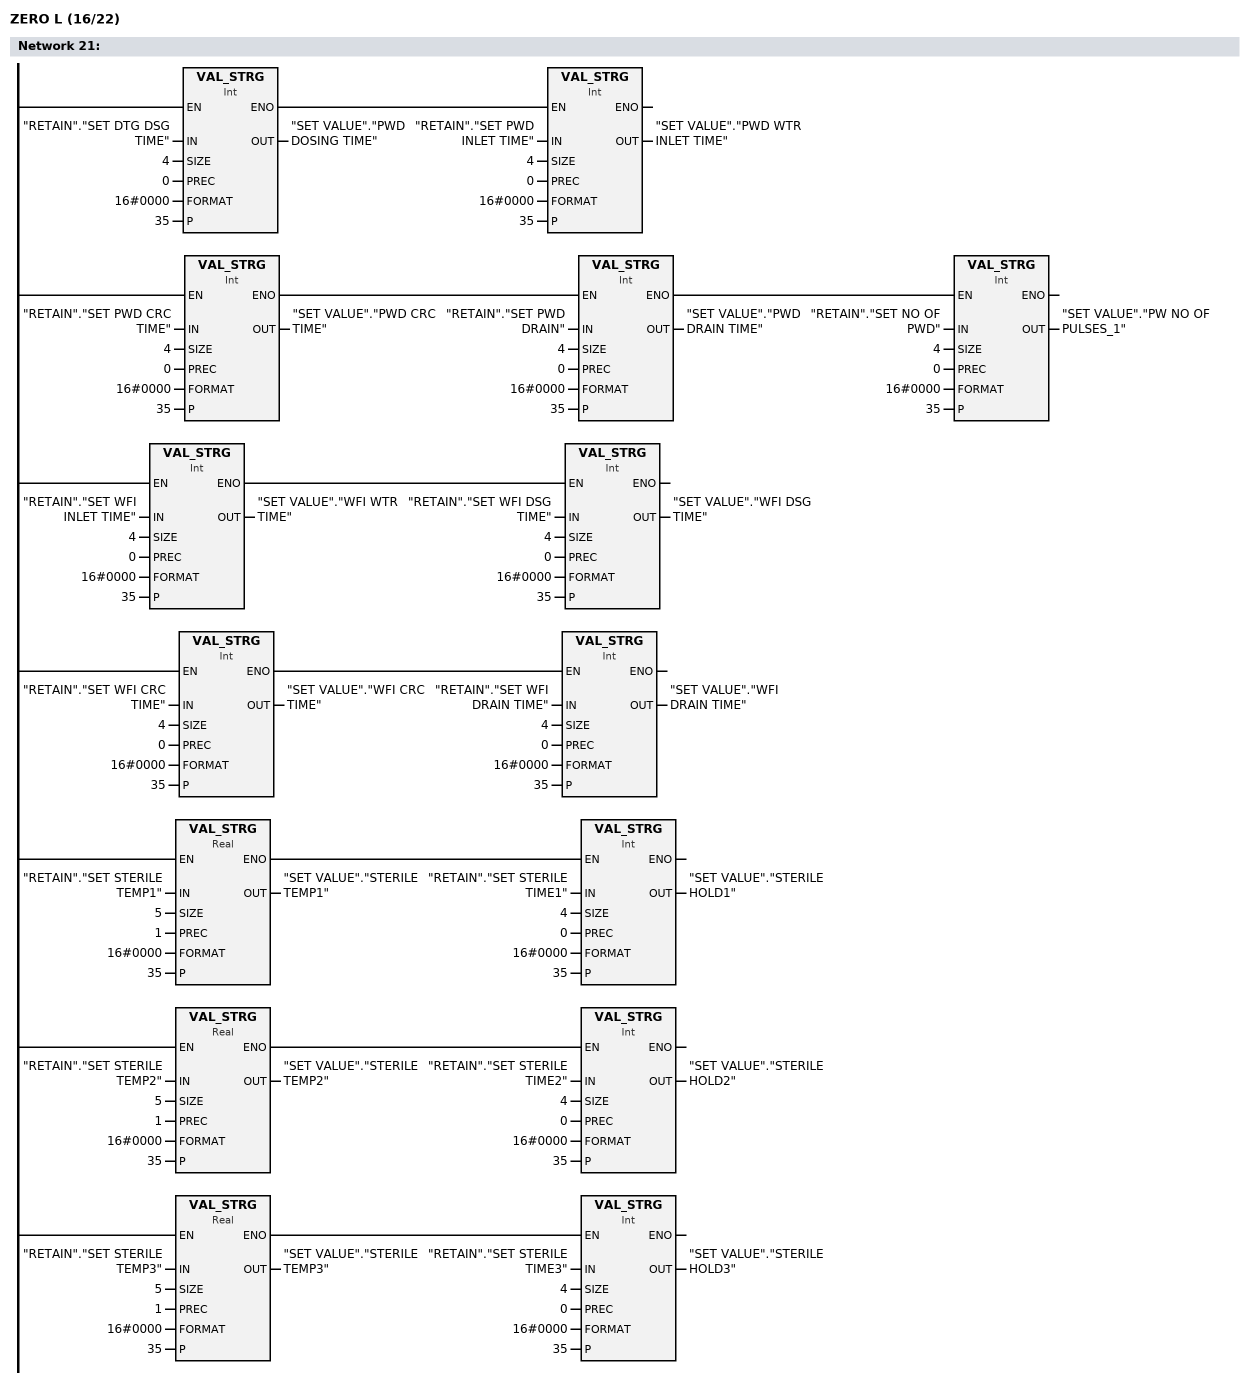
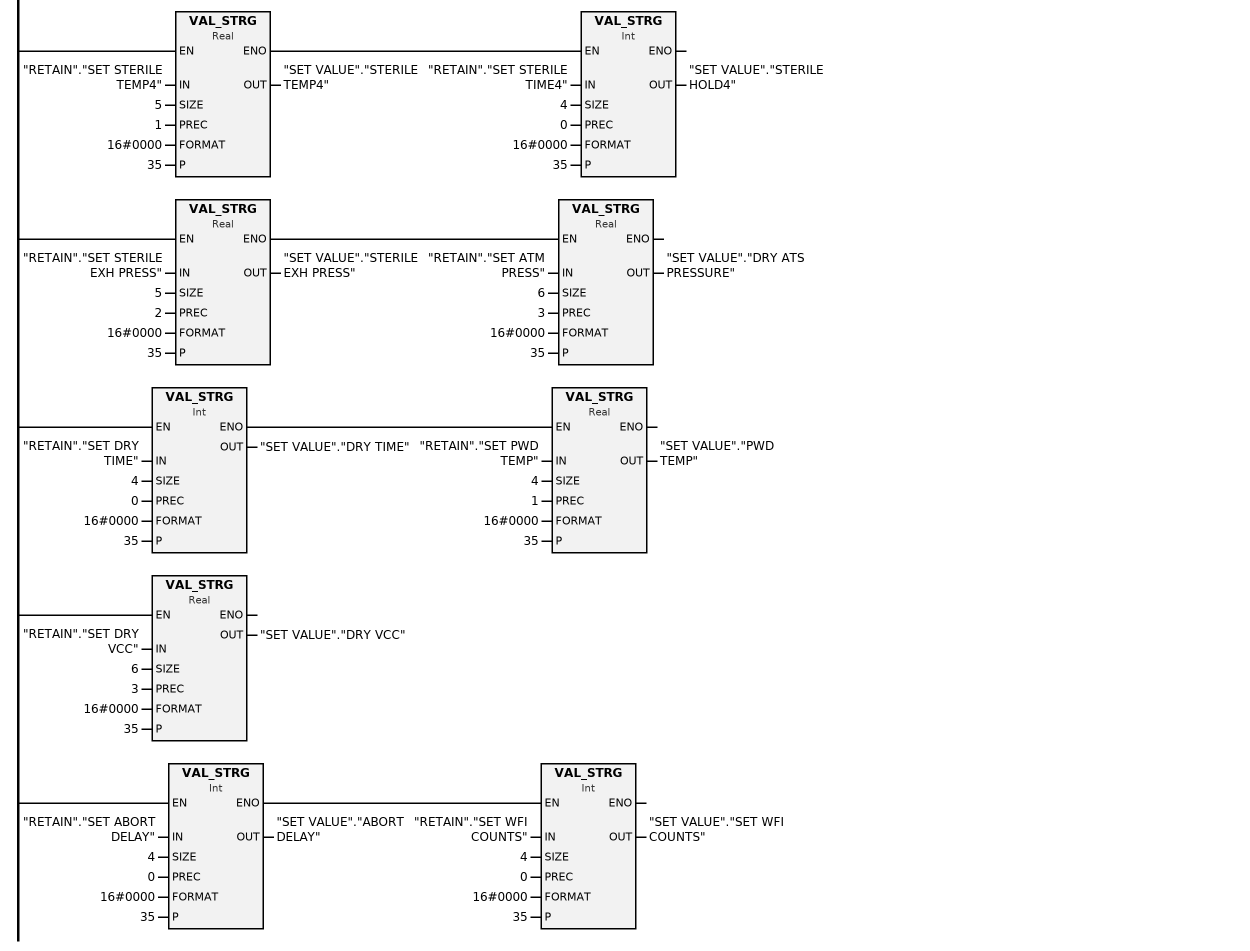
   RUNG wire#powerrail
      { S7_Templates := "[value_type := Int, str_type := String]" } VAL_STRG(IN := "RETAIN"."SET DTG DSG TIME", SIZE := 4, PREC := 0, FORMAT := 16#0000, P := 35, OUT => "SET VALUE"."PWD DOSING TIME")
      { S7_Templates := "[value_type := Int, str_type := String]" } VAL_STRG(IN := "RETAIN"."SET PWD INLET TIME", SIZE := 4, PREC := 0, FORMAT := 16#0000, P := 35, OUT => "SET VALUE"."PWD WTR INLET TIME")
   END_RUNG
   RUNG wire#powerrail
      { S7_Templates := "[value_type := Int, str_type := String]" } VAL_STRG(IN := "RETAIN"."SET PWD CRC TIME", SIZE := 4, PREC := 0, FORMAT := 16#0000, P := 35, OUT => "SET VALUE"."PWD CRC TIME")
      { S7_Templates := "[value_type := Int, str_type := String]" } VAL_STRG(IN := "RETAIN"."SET PWD DRAIN", SIZE := 4, PREC := 0, FORMAT := 16#0000, P := 35, OUT => "SET VALUE"."PWD DRAIN TIME")
      { S7_Templates := "[value_type := Int, str_type := String]" } VAL_STRG(IN := "RETAIN"."SET NO OF PWD", SIZE := 4, PREC := 0, FORMAT := 16#0000, P := 35, OUT => "SET VALUE"."PW NO OF PULSES_1")
   END_RUNG
   RUNG wire#powerrail
      { S7_Templates := "[value_type := Int, str_type := String]" } VAL_STRG(IN := "RETAIN"."SET WFI INLET TIME", SIZE := 4, PREC := 0, FORMAT := 16#0000, P := 35, OUT => "SET VALUE"."WFI WTR TIME")
      { S7_Templates := "[value_type := Int, str_type := String]" } VAL_STRG(IN := "RETAIN"."SET WFI DSG TIME", SIZE := 4, PREC := 0, FORMAT := 16#0000, P := 35, OUT => "SET VALUE"."WFI DSG TIME")
   END_RUNG
   RUNG wire#powerrail
      { S7_Templates := "[value_type := Int, str_type := String]" } VAL_STRG(IN := "RETAIN"."SET WFI CRC TIME", SIZE := 4, PREC := 0, FORMAT := 16#0000, P := 35, OUT => "SET VALUE"."WFI CRC TIME")
      { S7_Templates := "[value_type := Int, str_type := String]" } VAL_STRG(IN := "RETAIN"."SET WFI DRAIN TIME", SIZE := 4, PREC := 0, FORMAT := 16#0000, P := 35, OUT => "SET VALUE"."WFI DRAIN TIME")
   END_RUNG
   RUNG wire#powerrail
      { S7_Templates := "[value_type := Real, str_type := String]" } VAL_STRG(IN := "RETAIN"."SET STERILE TEMP1", SIZE := 5, PREC := 1, FORMAT := 16#0000, P := 35, OUT => "SET VALUE"."STERILE TEMP1")
      { S7_Templates := "[value_type := Int, str_type := String]" } VAL_STRG(IN := "RETAIN"."SET STERILE TIME1", SIZE := 4, PREC := 0, FORMAT := 16#0000, P := 35, OUT => "SET VALUE"."STERILE HOLD1")
   END_RUNG
   RUNG wire#powerrail
      { S7_Templates := "[value_type := Real, str_type := String]" } VAL_STRG(IN := "RETAIN"."SET STERILE TEMP2", SIZE := 5, PREC := 1, FORMAT := 16#0000, P := 35, OUT => "SET VALUE"."STERILE TEMP2")
      { S7_Templates := "[value_type := Int, str_type := String]" } VAL_STRG(IN := "RETAIN"."SET STERILE TIME2", SIZE := 4, PREC := 0, FORMAT := 16#0000, P := 35, OUT => "SET VALUE"."STERILE HOLD2")
   END_RUNG
   RUNG wire#powerrail
      { S7_Templates := "[value_type := Real, str_type := String]" } VAL_STRG(IN := "RETAIN"."SET STERILE TEMP3", SIZE := 5, PREC := 1, FORMAT := 16#0000, P := 35, OUT => "SET VALUE"."STERILE TEMP3")
      { S7_Templates := "[value_type := Int, str_type := String]" } VAL_STRG(IN := "RETAIN"."SET STERILE TIME3", SIZE := 4, PREC := 0, FORMAT := 16#0000, P := 35, OUT => "SET VALUE"."STERILE HOLD3")
   END_RUNG
   RUNG wire#powerrail
      { S7_Templates := "[value_type := Real, str_type := String]" } VAL_STRG(IN := "RETAIN"."SET STERILE TEMP4", SIZE := 5, PREC := 1, FORMAT := 16#0000, P := 35, OUT => "SET VALUE"."STERILE TEMP4")
      { S7_Templates := "[value_type := Int, str_type := String]" } VAL_STRG(IN := "RETAIN"."SET STERILE TIME4", SIZE := 4, PREC := 0, FORMAT := 16#0000, P := 35, OUT => "SET VALUE"."STERILE HOLD4")
   END_RUNG
   RUNG wire#powerrail
      { S7_Templates := "[value_type := Real, str_type := String]" } VAL_STRG(IN := "RETAIN"."SET STERILE EXH PRESS", SIZE := 5, PREC := 2, FORMAT := 16#0000, P := 35, OUT => "SET VALUE"."STERILE EXH PRESS")
      { S7_Templates := "[value_type := Real, str_type := String]" } VAL_STRG(IN := "RETAIN"."SET ATM PRESS", SIZE := 6, PREC := 3, FORMAT := 16#0000, P := 35, OUT => "SET VALUE"."DRY ATS PRESSURE")
   END_RUNG
   RUNG wire#powerrail
      { S7_Templates := "[value_type := Int, str_type := String]" } VAL_STRG(IN := "RETAIN"."SET DRY TIME", SIZE := 4, PREC := 0, FORMAT := 16#0000, P := 35, OUT => "SET VALUE"."DRY TIME")
      { S7_Templates := "[value_type := Real, str_type := String]" } VAL_STRG(IN := "RETAIN"."SET PWD TEMP", SIZE := 4, PREC := 1, FORMAT := 16#0000, P := 35, OUT => "SET VALUE"."PWD TEMP")
   END_RUNG
   RUNG wire#powerrail
      { S7_Templates := "[value_type := Real, str_type := String]" } VAL_STRG(IN := "RETAIN"."SET DRY VCC", SIZE := 6, PREC := 3, FORMAT := 16#0000, P := 35, OUT => "SET VALUE"."DRY VCC")
   END_RUNG
   RUNG wire#powerrail
      { S7_Templates := "[value_type := Int, str_type := String]" } VAL_STRG(IN := "RETAIN"."SET ABORT DELAY", SIZE := 4, PREC := 0, FORMAT := 16#0000, P := 35, OUT => "SET VALUE"."ABORT DELAY")
      { S7_Templates := "[value_type := Int, str_type := String]" } VAL_STRG(IN := "RETAIN"."SET WFI COUNTS", SIZE := 4, PREC := 0, FORMAT := 16#0000, P := 35, OUT => "SET VALUE"."SET WFI COUNTS")
   END_RUNG
   // the same network as SCL:
   VAL_STRG(IN := "RETAIN"."SET DTG DSG TIME",
            SIZE := 4,
            PREC := 0,
            FORMAT := 16#0000,
            P := 35,
            OUT => "SET VALUE"."PWD DOSING TIME",
            ENO => #_w1);
   IF #_w1 THEN
       VAL_STRG(IN := "RETAIN"."SET PWD INLET TIME",
                SIZE := 4,
                PREC := 0,
                FORMAT := 16#0000,
                P := 35,
                OUT => "SET VALUE"."PWD WTR INLET TIME");
   END_IF;
   VAL_STRG(IN := "RETAIN"."SET PWD CRC TIME",
            SIZE := 4,
            PREC := 0,
            FORMAT := 16#0000,
            P := 35,
            OUT => "SET VALUE"."PWD CRC TIME",
            ENO => #_w2);
   VAL_STRG(EN := #_w2,
            IN := "RETAIN"."SET PWD DRAIN",
            SIZE := 4,
            PREC := 0,
            FORMAT := 16#0000,
            P := 35,
            OUT => "SET VALUE"."PWD DRAIN TIME",
            ENO => #_w3);
   IF #_w3 THEN
       VAL_STRG(IN := "RETAIN"."SET NO OF PWD",
                SIZE := 4,
                PREC := 0,
                FORMAT := 16#0000,
                P := 35,
                OUT => "SET VALUE"."PW NO OF PULSES_1");
   END_IF;
   VAL_STRG(IN := "RETAIN"."SET WFI INLET TIME",
            SIZE := 4,
            PREC := 0,
            FORMAT := 16#0000,
            P := 35,
            OUT => "SET VALUE"."WFI WTR TIME",
            ENO => #_w4);
   IF #_w4 THEN
       VAL_STRG(IN := "RETAIN"."SET WFI DSG TIME",
                SIZE := 4,
                PREC := 0,
                FORMAT := 16#0000,
                P := 35,
                OUT => "SET VALUE"."WFI DSG TIME");
   END_IF;
   VAL_STRG(IN := "RETAIN"."SET WFI CRC TIME",
            SIZE := 4,
            PREC := 0,
            FORMAT := 16#0000,
            P := 35,
            OUT => "SET VALUE"."WFI CRC TIME",
            ENO => #_w5);
   IF #_w5 THEN
       VAL_STRG(IN := "RETAIN"."SET WFI DRAIN TIME",
                SIZE := 4,
                PREC := 0,
                FORMAT := 16#0000,
                P := 35,
                OUT => "SET VALUE"."WFI DRAIN TIME");
   END_IF;
   VAL_STRG(IN := "RETAIN"."SET STERILE TEMP1",
            SIZE := 5,
            PREC := 1,
            FORMAT := 16#0000,
            P := 35,
            OUT => "SET VALUE"."STERILE TEMP1",
            ENO => #_w6);
   IF #_w6 THEN
       VAL_STRG(IN := "RETAIN"."SET STERILE TIME1",
                SIZE := 4,
                PREC := 0,
                FORMAT := 16#0000,
                P := 35,
                OUT => "SET VALUE"."STERILE HOLD1");
   END_IF;
   VAL_STRG(IN := "RETAIN"."SET STERILE TEMP2",
            SIZE := 5,
            PREC := 1,
            FORMAT := 16#0000,
            P := 35,
            OUT => "SET VALUE"."STERILE TEMP2",
            ENO => #_w7);
   IF #_w7 THEN
       VAL_STRG(IN := "RETAIN"."SET STERILE TIME2",
                SIZE := 4,
                PREC := 0,
                FORMAT := 16#0000,
                P := 35,
                OUT => "SET VALUE"."STERILE HOLD2");
   END_IF;
   VAL_STRG(IN := "RETAIN"."SET STERILE TEMP3",
            SIZE := 5,
            PREC := 1,
            FORMAT := 16#0000,
            P := 35,
            OUT => "SET VALUE"."STERILE TEMP3",
            ENO => #_w8);
   IF #_w8 THEN
       VAL_STRG(IN := "RETAIN"."SET STERILE TIME3",
                SIZE := 4,
                PREC := 0,
                FORMAT := 16#0000,
                P := 35,
                OUT => "SET VALUE"."STERILE HOLD3");
   END_IF;
   VAL_STRG(IN := "RETAIN"."SET STERILE TEMP4",
            SIZE := 5,
            PREC := 1,
            FORMAT := 16#0000,
            P := 35,
            OUT => "SET VALUE"."STERILE TEMP4",
            ENO => #_w9);
   IF #_w9 THEN
       VAL_STRG(IN := "RETAIN"."SET STERILE TIME4",
                SIZE := 4,
                PREC := 0,
                FORMAT := 16#0000,
                P := 35,
                OUT => "SET VALUE"."STERILE HOLD4");
   END_IF;
   VAL_STRG(IN := "RETAIN"."SET STERILE EXH PRESS",
            SIZE := 5,
            PREC := 2,
            FORMAT := 16#0000,
            P := 35,
            OUT => "SET VALUE"."STERILE EXH PRESS",
            ENO => #_w10);
   IF #_w10 THEN
       VAL_STRG(IN := "RETAIN"."SET ATM PRESS",
                SIZE := 6,
                PREC := 3,
                FORMAT := 16#0000,
                P := 35,
                OUT => "SET VALUE"."DRY ATS PRESSURE");
   END_IF;
   VAL_STRG(IN := "RETAIN"."SET DRY TIME",
            SIZE := 4,
            PREC := 0,
            FORMAT := 16#0000,
            P := 35,
            OUT => "SET VALUE"."DRY TIME",
            ENO => #_w11);
   IF #_w11 THEN
       VAL_STRG(IN := "RETAIN"."SET PWD TEMP",
                SIZE := 4,
                PREC := 1,
                FORMAT := 16#0000,
                P := 35,
                OUT => "SET VALUE"."PWD TEMP");
   END_IF;
   VAL_STRG(IN := "RETAIN"."SET DRY VCC",
            SIZE := 6,
            PREC := 3,
            FORMAT := 16#0000,
            P := 35,
            OUT => "SET VALUE"."DRY VCC");
   VAL_STRG(IN := "RETAIN"."SET ABORT DELAY",
            SIZE := 4,
            PREC := 0,
            FORMAT := 16#0000,
            P := 35,
            OUT => "SET VALUE"."ABORT DELAY",
            ENO => #_w12);
   IF #_w12 THEN
       VAL_STRG(IN := "RETAIN"."SET WFI COUNTS",
                SIZE := 4,
                PREC := 0,
                FORMAT := 16#0000,
                P := 35,
                OUT => "SET VALUE"."SET WFI COUNTS");
   END_IF;
END_REGION

REGION Network 22
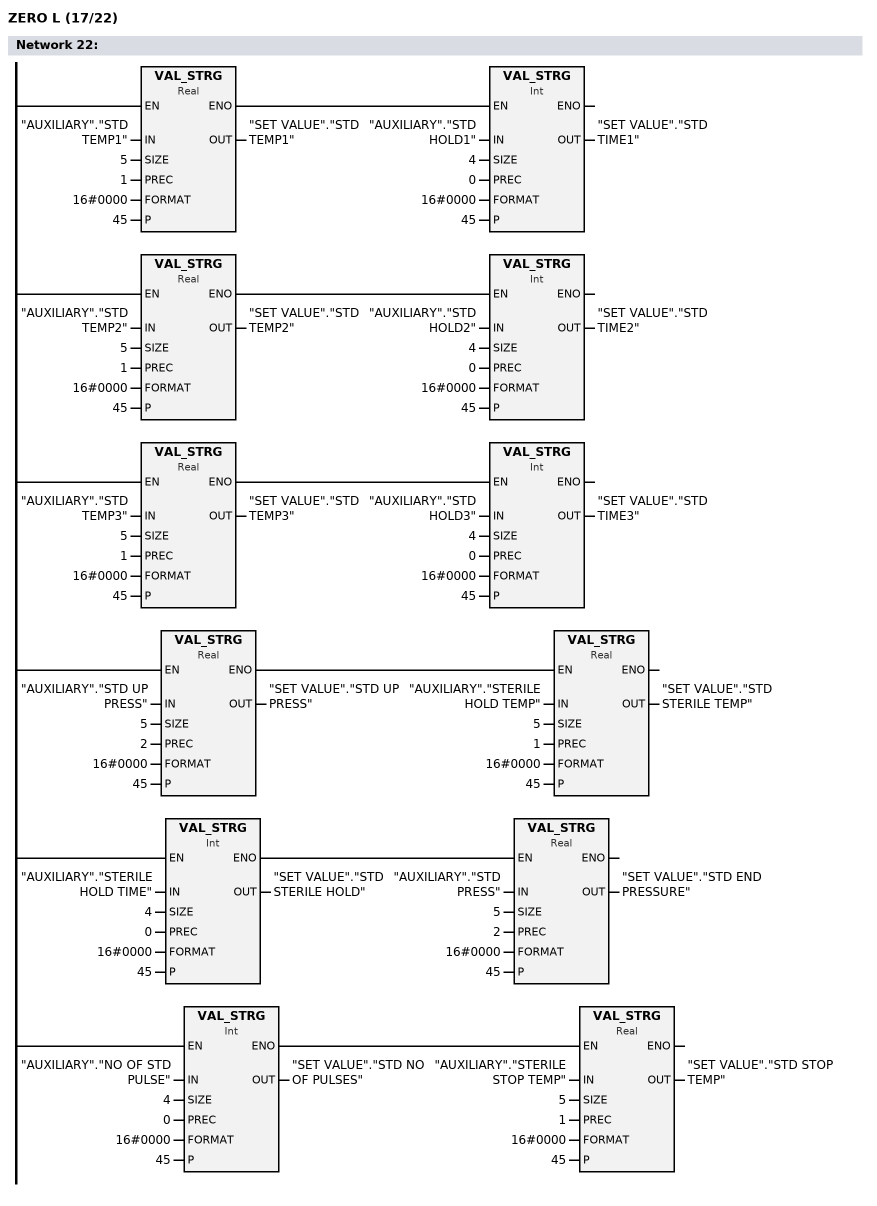
   RUNG wire#powerrail
      { S7_Templates := "[value_type := Real, str_type := String]" } VAL_STRG(IN := "AUXILIARY"."STD TEMP1", SIZE := 5, PREC := 1, FORMAT := 16#0000, P := 45, OUT => "SET VALUE"."STD TEMP1")
      { S7_Templates := "[value_type := Int, str_type := String]" } VAL_STRG(IN := "AUXILIARY"."STD HOLD1", SIZE := 4, PREC := 0, FORMAT := 16#0000, P := 45, OUT => "SET VALUE"."STD TIME1")
   END_RUNG
   RUNG wire#powerrail
      { S7_Templates := "[value_type := Real, str_type := String]" } VAL_STRG(IN := "AUXILIARY"."STD TEMP2", SIZE := 5, PREC := 1, FORMAT := 16#0000, P := 45, OUT => "SET VALUE"."STD TEMP2")
      { S7_Templates := "[value_type := Int, str_type := String]" } VAL_STRG(IN := "AUXILIARY"."STD HOLD2", SIZE := 4, PREC := 0, FORMAT := 16#0000, P := 45, OUT => "SET VALUE"."STD TIME2")
   END_RUNG
   RUNG wire#powerrail
      { S7_Templates := "[value_type := Real, str_type := String]" } VAL_STRG(IN := "AUXILIARY"."STD TEMP3", SIZE := 5, PREC := 1, FORMAT := 16#0000, P := 45, OUT => "SET VALUE"."STD TEMP3")
      { S7_Templates := "[value_type := Int, str_type := String]" } VAL_STRG(IN := "AUXILIARY"."STD HOLD3", SIZE := 4, PREC := 0, FORMAT := 16#0000, P := 45, OUT => "SET VALUE"."STD TIME3")
   END_RUNG
   RUNG wire#powerrail
      { S7_Templates := "[value_type := Real, str_type := String]" } VAL_STRG(IN := "AUXILIARY"."STD UP PRESS", SIZE := 5, PREC := 2, FORMAT := 16#0000, P := 45, OUT => "SET VALUE"."STD UP PRESS")
      { S7_Templates := "[value_type := Real, str_type := String]" } VAL_STRG(IN := "AUXILIARY"."STERILE HOLD TEMP", SIZE := 5, PREC := 1, FORMAT := 16#0000, P := 45, OUT => "SET VALUE"."STD STERILE TEMP")
   END_RUNG
   RUNG wire#powerrail
      { S7_Templates := "[value_type := Int, str_type := String]" } VAL_STRG(IN := "AUXILIARY"."STERILE HOLD TIME", SIZE := 4, PREC := 0, FORMAT := 16#0000, P := 45, OUT => "SET VALUE"."STD STERILE HOLD")
      { S7_Templates := "[value_type := Real, str_type := String]" } VAL_STRG(IN := "AUXILIARY"."STD PRESS", SIZE := 5, PREC := 2, FORMAT := 16#0000, P := 45, OUT => "SET VALUE"."STD END PRESSURE")
   END_RUNG
   RUNG wire#powerrail
      { S7_Templates := "[value_type := Int, str_type := String]" } VAL_STRG(IN := "AUXILIARY"."NO OF STD PULSE", SIZE := 4, PREC := 0, FORMAT := 16#0000, P := 45, OUT => "SET VALUE"."STD NO OF PULSES")
      { S7_Templates := "[value_type := Real, str_type := String]" } VAL_STRG(IN := "AUXILIARY"."STERILE STOP TEMP", SIZE := 5, PREC := 1, FORMAT := 16#0000, P := 45, OUT => "SET VALUE"."STD STOP TEMP")
   END_RUNG
   // the same network as SCL:
   VAL_STRG(IN := "AUXILIARY"."STD TEMP1",
            SIZE := 5,
            PREC := 1,
            FORMAT := 16#0000,
            P := 45,
            OUT => "SET VALUE"."STD TEMP1",
            ENO => #_w1);
   IF #_w1 THEN
       VAL_STRG(IN := "AUXILIARY"."STD HOLD1",
                SIZE := 4,
                PREC := 0,
                FORMAT := 16#0000,
                P := 45,
                OUT => "SET VALUE"."STD TIME1");
   END_IF;
   VAL_STRG(IN := "AUXILIARY"."STD TEMP2",
            SIZE := 5,
            PREC := 1,
            FORMAT := 16#0000,
            P := 45,
            OUT => "SET VALUE"."STD TEMP2",
            ENO => #_w2);
   IF #_w2 THEN
       VAL_STRG(IN := "AUXILIARY"."STD HOLD2",
                SIZE := 4,
                PREC := 0,
                FORMAT := 16#0000,
                P := 45,
                OUT => "SET VALUE"."STD TIME2");
   END_IF;
   VAL_STRG(IN := "AUXILIARY"."STD TEMP3",
            SIZE := 5,
            PREC := 1,
            FORMAT := 16#0000,
            P := 45,
            OUT => "SET VALUE"."STD TEMP3",
            ENO => #_w3);
   IF #_w3 THEN
       VAL_STRG(IN := "AUXILIARY"."STD HOLD3",
                SIZE := 4,
                PREC := 0,
                FORMAT := 16#0000,
                P := 45,
                OUT => "SET VALUE"."STD TIME3");
   END_IF;
   VAL_STRG(IN := "AUXILIARY"."STD UP PRESS",
            SIZE := 5,
            PREC := 2,
            FORMAT := 16#0000,
            P := 45,
            OUT => "SET VALUE"."STD UP PRESS",
            ENO => #_w4);
   IF #_w4 THEN
       VAL_STRG(IN := "AUXILIARY"."STERILE HOLD TEMP",
                SIZE := 5,
                PREC := 1,
                FORMAT := 16#0000,
                P := 45,
                OUT => "SET VALUE"."STD STERILE TEMP");
   END_IF;
   VAL_STRG(IN := "AUXILIARY"."STERILE HOLD TIME",
            SIZE := 4,
            PREC := 0,
            FORMAT := 16#0000,
            P := 45,
            OUT => "SET VALUE"."STD STERILE HOLD",
            ENO => #_w5);
   IF #_w5 THEN
       VAL_STRG(IN := "AUXILIARY"."STD PRESS",
                SIZE := 5,
                PREC := 2,
                FORMAT := 16#0000,
                P := 45,
                OUT => "SET VALUE"."STD END PRESSURE");
   END_IF;
   VAL_STRG(IN := "AUXILIARY"."NO OF STD PULSE",
            SIZE := 4,
            PREC := 0,
            FORMAT := 16#0000,
            P := 45,
            OUT => "SET VALUE"."STD NO OF PULSES",
            ENO => #_w6);
   IF #_w6 THEN
       VAL_STRG(IN := "AUXILIARY"."STERILE STOP TEMP",
                SIZE := 5,
                PREC := 1,
                FORMAT := 16#0000,
                P := 45,
                OUT => "SET VALUE"."STD STOP TEMP");
   END_IF;
END_REGION

REGION Network 23
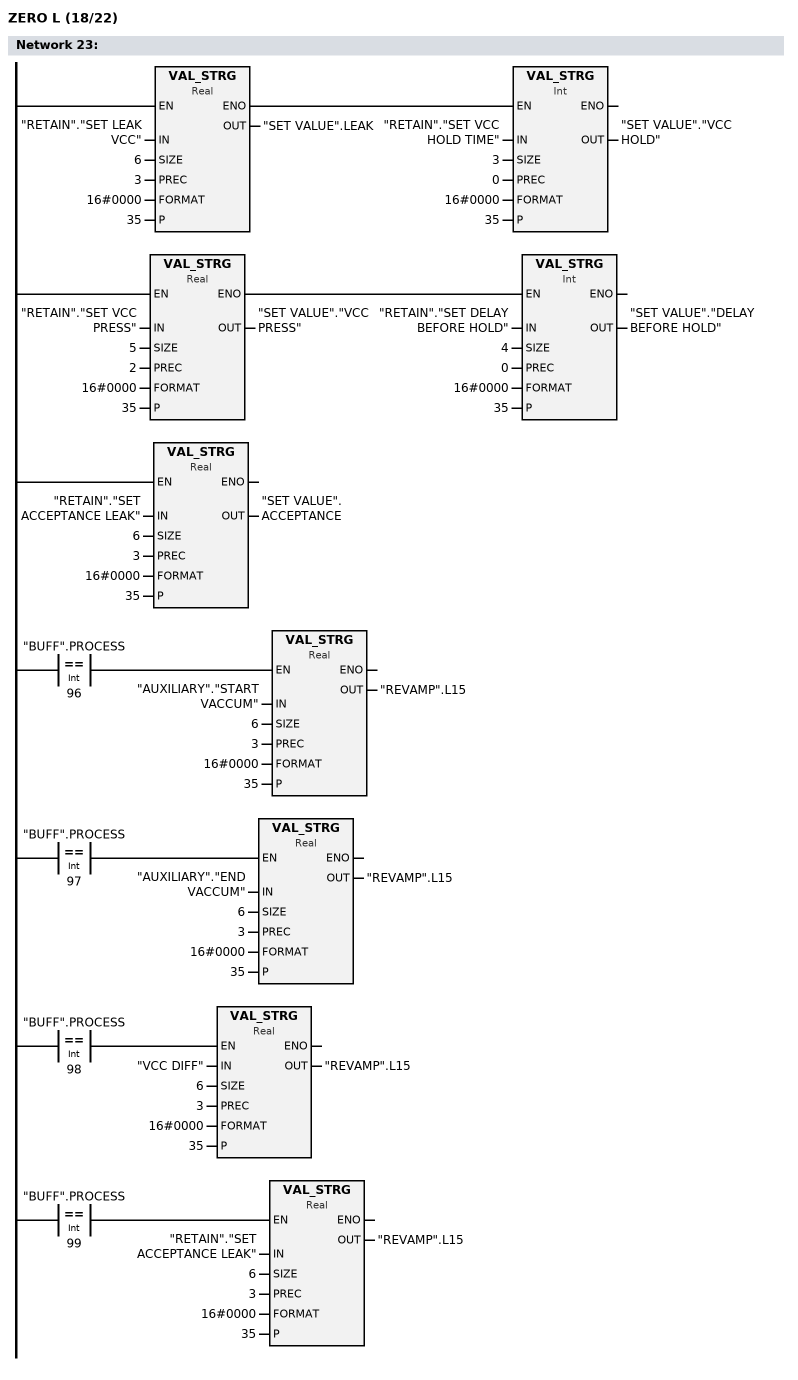
   RUNG wire#powerrail
      { S7_Templates := "[value_type := Real, str_type := String]" } VAL_STRG(IN := "RETAIN"."SET LEAK VCC", SIZE := 6, PREC := 3, FORMAT := 16#0000, P := 35, OUT => "SET VALUE".LEAK)
      { S7_Templates := "[value_type := Int, str_type := String]" } VAL_STRG(IN := "RETAIN"."SET VCC HOLD TIME", SIZE := 3, PREC := 0, FORMAT := 16#0000, P := 35, OUT => "SET VALUE"."VCC HOLD")
   END_RUNG
   RUNG wire#powerrail
      { S7_Templates := "[value_type := Real, str_type := String]" } VAL_STRG(IN := "RETAIN"."SET VCC PRESS", SIZE := 5, PREC := 2, FORMAT := 16#0000, P := 35, OUT => "SET VALUE"."VCC PRESS")
      { S7_Templates := "[value_type := Int, str_type := String]" } VAL_STRG(IN := "RETAIN"."SET DELAY BEFORE HOLD", SIZE := 4, PREC := 0, FORMAT := 16#0000, P := 35, OUT => "SET VALUE"."DELAY BEFORE HOLD")
   END_RUNG
   RUNG wire#powerrail
      { S7_Templates := "[value_type := Real, str_type := String]" } VAL_STRG(IN := "RETAIN"."SET ACCEPTANCE LEAK", SIZE := 6, PREC := 3, FORMAT := 16#0000, P := 35, OUT => "SET VALUE".ACCEPTANCE)
   END_RUNG
   RUNG wire#powerrail
      { S7_Templates := "SrcType := Int" } EQ_Contact(in1 := "BUFF".PROCESS, in2 := 96)
      { S7_Templates := "[value_type := Real, str_type := String]" } VAL_STRG(IN := "AUXILIARY"."START VACCUM", SIZE := 6, PREC := 3, FORMAT := 16#0000, P := 35, OUT => "REVAMP".L15)
   END_RUNG
   RUNG wire#powerrail
      { S7_Templates := "SrcType := Int" } EQ_Contact(in1 := "BUFF".PROCESS, in2 := 97)
      { S7_Templates := "[value_type := Real, str_type := String]" } VAL_STRG(IN := "AUXILIARY"."END VACCUM", SIZE := 6, PREC := 3, FORMAT := 16#0000, P := 35, OUT => "REVAMP".L15)
   END_RUNG
   RUNG wire#powerrail
      { S7_Templates := "SrcType := Int" } EQ_Contact(in1 := "BUFF".PROCESS, in2 := 98)
      { S7_Templates := "[value_type := Real, str_type := String]" } VAL_STRG(IN := "VCC DIFF", SIZE := 6, PREC := 3, FORMAT := 16#0000, P := 35, OUT => "REVAMP".L15)
   END_RUNG
   RUNG wire#powerrail
      { S7_Templates := "SrcType := Int" } EQ_Contact(in1 := "BUFF".PROCESS, in2 := 99)
      { S7_Templates := "[value_type := Real, str_type := String]" } VAL_STRG(IN := "RETAIN"."SET ACCEPTANCE LEAK", SIZE := 6, PREC := 3, FORMAT := 16#0000, P := 35, OUT => "REVAMP".L15)
   END_RUNG
   // the same network as SCL:
   VAL_STRG(IN := "RETAIN"."SET LEAK VCC",
            SIZE := 6,
            PREC := 3,
            FORMAT := 16#0000,
            P := 35,
            OUT => "SET VALUE".LEAK,
            ENO => #_w1);
   IF #_w1 THEN
       VAL_STRG(IN := "RETAIN"."SET VCC HOLD TIME",
                SIZE := 3,
                PREC := 0,
                FORMAT := 16#0000,
                P := 35,
                OUT => "SET VALUE"."VCC HOLD");
   END_IF;
   VAL_STRG(IN := "RETAIN"."SET VCC PRESS",
            SIZE := 5,
            PREC := 2,
            FORMAT := 16#0000,
            P := 35,
            OUT => "SET VALUE"."VCC PRESS",
            ENO => #_w2);
   IF #_w2 THEN
       VAL_STRG(IN := "RETAIN"."SET DELAY BEFORE HOLD",
                SIZE := 4,
                PREC := 0,
                FORMAT := 16#0000,
                P := 35,
                OUT => "SET VALUE"."DELAY BEFORE HOLD");
   END_IF;
   VAL_STRG(IN := "RETAIN"."SET ACCEPTANCE LEAK",
            SIZE := 6,
            PREC := 3,
            FORMAT := 16#0000,
            P := 35,
            OUT => "SET VALUE".ACCEPTANCE);
   IF "BUFF".PROCESS = 96 THEN
       VAL_STRG(IN := "AUXILIARY"."START VACCUM",
                SIZE := 6,
                PREC := 3,
                FORMAT := 16#0000,
                P := 35,
                OUT => "REVAMP".L15);
   END_IF;
   IF "BUFF".PROCESS = 97 THEN
       VAL_STRG(IN := "AUXILIARY"."END VACCUM",
                SIZE := 6,
                PREC := 3,
                FORMAT := 16#0000,
                P := 35,
                OUT => "REVAMP".L15);
   END_IF;
   IF "BUFF".PROCESS = 98 THEN
       VAL_STRG(IN := "VCC DIFF", SIZE := 6, PREC := 3, FORMAT := 16#0000, P := 35, OUT => "REVAMP".L15);
   END_IF;
   IF "BUFF".PROCESS = 99 THEN
       VAL_STRG(IN := "RETAIN"."SET ACCEPTANCE LEAK",
                SIZE := 6,
                PREC := 3,
                FORMAT := 16#0000,
                P := 35,
                OUT => "REVAMP".L15);
   END_IF;
END_REGION

REGION Network 24
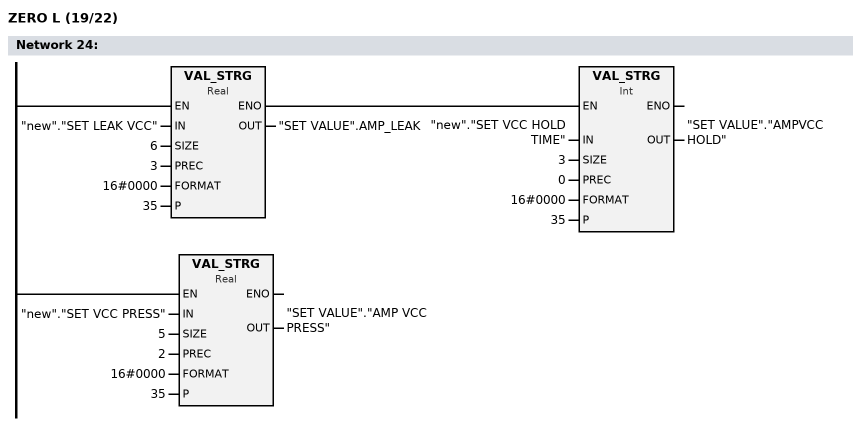
   RUNG wire#powerrail
      { S7_Templates := "[value_type := Real, str_type := String]" } VAL_STRG(IN := "new"."SET LEAK VCC", SIZE := 6, PREC := 3, FORMAT := 16#0000, P := 35, OUT => "SET VALUE".AMP_LEAK)
      { S7_Templates := "[value_type := Int, str_type := String]" } VAL_STRG(IN := "new"."SET VCC HOLD TIME", SIZE := 3, PREC := 0, FORMAT := 16#0000, P := 35, OUT => "SET VALUE"."AMPVCC HOLD")
   END_RUNG
   RUNG wire#powerrail
      { S7_Templates := "[value_type := Real, str_type := String]" } VAL_STRG(IN := "new"."SET VCC PRESS", SIZE := 5, PREC := 2, FORMAT := 16#0000, P := 35, OUT => "SET VALUE"."AMP VCC PRESS")
   END_RUNG
   // the same network as SCL:
   VAL_STRG(IN := "new"."SET LEAK VCC",
            SIZE := 6,
            PREC := 3,
            FORMAT := 16#0000,
            P := 35,
            OUT => "SET VALUE".AMP_LEAK,
            ENO => #_w1);
   IF #_w1 THEN
       VAL_STRG(IN := "new"."SET VCC HOLD TIME",
                SIZE := 3,
                PREC := 0,
                FORMAT := 16#0000,
                P := 35,
                OUT => "SET VALUE"."AMPVCC HOLD");
   END_IF;
   VAL_STRG(IN := "new"."SET VCC PRESS",
            SIZE := 5,
            PREC := 2,
            FORMAT := 16#0000,
            P := 35,
            OUT => "SET VALUE"."AMP VCC PRESS");
END_REGION

REGION Network 25
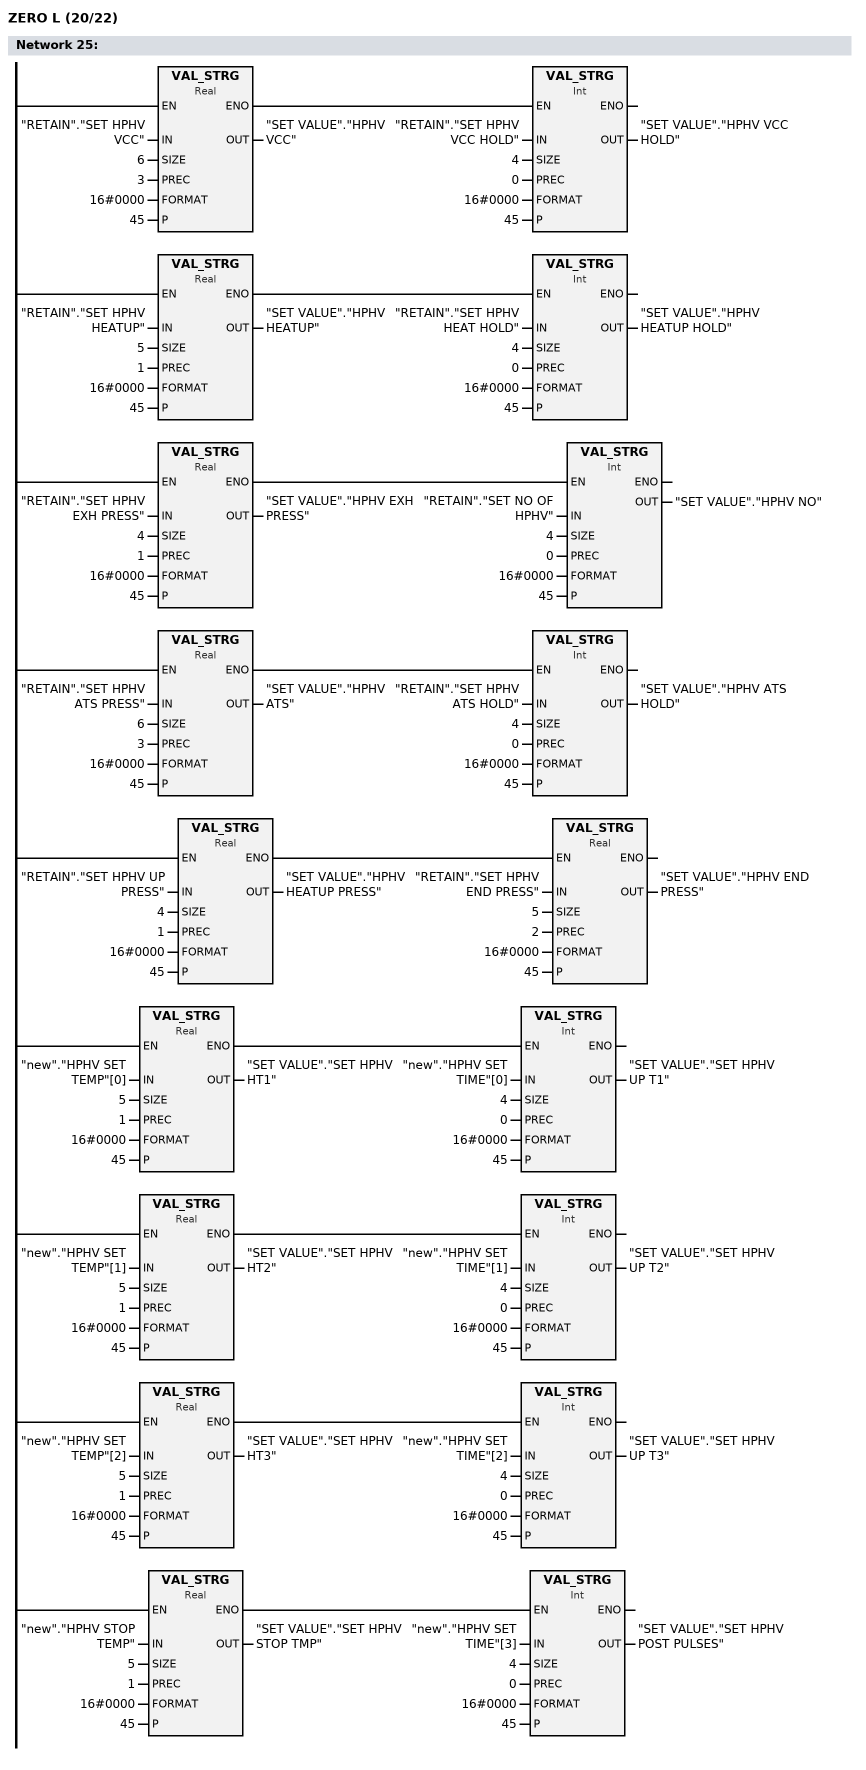
   RUNG wire#powerrail
      { S7_Templates := "[value_type := Real, str_type := String]" } VAL_STRG(IN := "RETAIN"."SET HPHV VCC", SIZE := 6, PREC := 3, FORMAT := 16#0000, P := 45, OUT => "SET VALUE"."HPHV VCC")
      { S7_Templates := "[value_type := Int, str_type := String]" } VAL_STRG(IN := "RETAIN"."SET HPHV VCC HOLD", SIZE := 4, PREC := 0, FORMAT := 16#0000, P := 45, OUT => "SET VALUE"."HPHV VCC HOLD")
   END_RUNG
   RUNG wire#powerrail
      { S7_Templates := "[value_type := Real, str_type := String]" } VAL_STRG(IN := "RETAIN"."SET HPHV HEATUP", SIZE := 5, PREC := 1, FORMAT := 16#0000, P := 45, OUT => "SET VALUE"."HPHV HEATUP")
      { S7_Templates := "[value_type := Int, str_type := String]" } VAL_STRG(IN := "RETAIN"."SET HPHV HEAT HOLD", SIZE := 4, PREC := 0, FORMAT := 16#0000, P := 45, OUT => "SET VALUE"."HPHV HEATUP HOLD")
   END_RUNG
   RUNG wire#powerrail
      { S7_Templates := "[value_type := Real, str_type := String]" } VAL_STRG(IN := "RETAIN"."SET HPHV EXH PRESS", SIZE := 4, PREC := 1, FORMAT := 16#0000, P := 45, OUT => "SET VALUE"."HPHV EXH PRESS")
      { S7_Templates := "[value_type := Int, str_type := String]" } VAL_STRG(IN := "RETAIN"."SET NO OF HPHV", SIZE := 4, PREC := 0, FORMAT := 16#0000, P := 45, OUT => "SET VALUE"."HPHV NO")
   END_RUNG
   RUNG wire#powerrail
      { S7_Templates := "[value_type := Real, str_type := String]" } VAL_STRG(IN := "RETAIN"."SET HPHV ATS PRESS", SIZE := 6, PREC := 3, FORMAT := 16#0000, P := 45, OUT => "SET VALUE"."HPHV ATS")
      { S7_Templates := "[value_type := Int, str_type := String]" } VAL_STRG(IN := "RETAIN"."SET HPHV ATS HOLD", SIZE := 4, PREC := 0, FORMAT := 16#0000, P := 45, OUT => "SET VALUE"."HPHV ATS HOLD")
   END_RUNG
   RUNG wire#powerrail
      { S7_Templates := "[value_type := Real, str_type := String]" } VAL_STRG(IN := "RETAIN"."SET HPHV UP PRESS", SIZE := 4, PREC := 1, FORMAT := 16#0000, P := 45, OUT => "SET VALUE"."HPHV HEATUP PRESS")
      { S7_Templates := "[value_type := Real, str_type := String]" } VAL_STRG(IN := "RETAIN"."SET HPHV END PRESS", SIZE := 5, PREC := 2, FORMAT := 16#0000, P := 45, OUT => "SET VALUE"."HPHV END PRESS")
   END_RUNG
   RUNG wire#powerrail
      { S7_Templates := "[value_type := Real, str_type := String]" } VAL_STRG(IN := "new"."HPHV SET TEMP"[0], SIZE := 5, PREC := 1, FORMAT := 16#0000, P := 45, OUT => "SET VALUE"."SET HPHV HT1")
      { S7_Templates := "[value_type := Int, str_type := String]" } VAL_STRG(IN := "new"."HPHV SET TIME"[0], SIZE := 4, PREC := 0, FORMAT := 16#0000, P := 45, OUT => "SET VALUE"."SET HPHV UP T1")
   END_RUNG
   RUNG wire#powerrail
      { S7_Templates := "[value_type := Real, str_type := String]" } VAL_STRG(IN := "new"."HPHV SET TEMP"[1], SIZE := 5, PREC := 1, FORMAT := 16#0000, P := 45, OUT => "SET VALUE"."SET HPHV HT2")
      { S7_Templates := "[value_type := Int, str_type := String]" } VAL_STRG(IN := "new"."HPHV SET TIME"[1], SIZE := 4, PREC := 0, FORMAT := 16#0000, P := 45, OUT => "SET VALUE"."SET HPHV UP T2")
   END_RUNG
   RUNG wire#powerrail
      { S7_Templates := "[value_type := Real, str_type := String]" } VAL_STRG(IN := "new"."HPHV SET TEMP"[2], SIZE := 5, PREC := 1, FORMAT := 16#0000, P := 45, OUT => "SET VALUE"."SET HPHV HT3")
      { S7_Templates := "[value_type := Int, str_type := String]" } VAL_STRG(IN := "new"."HPHV SET TIME"[2], SIZE := 4, PREC := 0, FORMAT := 16#0000, P := 45, OUT => "SET VALUE"."SET HPHV UP T3")
   END_RUNG
   RUNG wire#powerrail
      { S7_Templates := "[value_type := Real, str_type := String]" } VAL_STRG(IN := "new"."HPHV STOP TEMP", SIZE := 5, PREC := 1, FORMAT := 16#0000, P := 45, OUT => "SET VALUE"."SET HPHV STOP TMP")
      { S7_Templates := "[value_type := Int, str_type := String]" } VAL_STRG(IN := "new"."HPHV SET TIME"[3], SIZE := 4, PREC := 0, FORMAT := 16#0000, P := 45, OUT => "SET VALUE"."SET HPHV POST PULSES")
   END_RUNG
   // the same network as SCL:
   VAL_STRG(IN := "RETAIN"."SET HPHV VCC",
            SIZE := 6,
            PREC := 3,
            FORMAT := 16#0000,
            P := 45,
            OUT => "SET VALUE"."HPHV VCC",
            ENO => #_w1);
   IF #_w1 THEN
       VAL_STRG(IN := "RETAIN"."SET HPHV VCC HOLD",
                SIZE := 4,
                PREC := 0,
                FORMAT := 16#0000,
                P := 45,
                OUT => "SET VALUE"."HPHV VCC HOLD");
   END_IF;
   VAL_STRG(IN := "RETAIN"."SET HPHV HEATUP",
            SIZE := 5,
            PREC := 1,
            FORMAT := 16#0000,
            P := 45,
            OUT => "SET VALUE"."HPHV HEATUP",
            ENO => #_w2);
   IF #_w2 THEN
       VAL_STRG(IN := "RETAIN"."SET HPHV HEAT HOLD",
                SIZE := 4,
                PREC := 0,
                FORMAT := 16#0000,
                P := 45,
                OUT => "SET VALUE"."HPHV HEATUP HOLD");
   END_IF;
   VAL_STRG(IN := "RETAIN"."SET HPHV EXH PRESS",
            SIZE := 4,
            PREC := 1,
            FORMAT := 16#0000,
            P := 45,
            OUT => "SET VALUE"."HPHV EXH PRESS",
            ENO => #_w3);
   IF #_w3 THEN
       VAL_STRG(IN := "RETAIN"."SET NO OF HPHV",
                SIZE := 4,
                PREC := 0,
                FORMAT := 16#0000,
                P := 45,
                OUT => "SET VALUE"."HPHV NO");
   END_IF;
   VAL_STRG(IN := "RETAIN"."SET HPHV ATS PRESS",
            SIZE := 6,
            PREC := 3,
            FORMAT := 16#0000,
            P := 45,
            OUT => "SET VALUE"."HPHV ATS",
            ENO => #_w4);
   IF #_w4 THEN
       VAL_STRG(IN := "RETAIN"."SET HPHV ATS HOLD",
                SIZE := 4,
                PREC := 0,
                FORMAT := 16#0000,
                P := 45,
                OUT => "SET VALUE"."HPHV ATS HOLD");
   END_IF;
   VAL_STRG(IN := "RETAIN"."SET HPHV UP PRESS",
            SIZE := 4,
            PREC := 1,
            FORMAT := 16#0000,
            P := 45,
            OUT => "SET VALUE"."HPHV HEATUP PRESS",
            ENO => #_w5);
   IF #_w5 THEN
       VAL_STRG(IN := "RETAIN"."SET HPHV END PRESS",
                SIZE := 5,
                PREC := 2,
                FORMAT := 16#0000,
                P := 45,
                OUT => "SET VALUE"."HPHV END PRESS");
   END_IF;
   VAL_STRG(IN := "new"."HPHV SET TEMP"[0],
            SIZE := 5,
            PREC := 1,
            FORMAT := 16#0000,
            P := 45,
            OUT => "SET VALUE"."SET HPHV HT1",
            ENO => #_w6);
   IF #_w6 THEN
       VAL_STRG(IN := "new"."HPHV SET TIME"[0],
                SIZE := 4,
                PREC := 0,
                FORMAT := 16#0000,
                P := 45,
                OUT => "SET VALUE"."SET HPHV UP T1");
   END_IF;
   VAL_STRG(IN := "new"."HPHV SET TEMP"[1],
            SIZE := 5,
            PREC := 1,
            FORMAT := 16#0000,
            P := 45,
            OUT => "SET VALUE"."SET HPHV HT2",
            ENO => #_w7);
   IF #_w7 THEN
       VAL_STRG(IN := "new"."HPHV SET TIME"[1],
                SIZE := 4,
                PREC := 0,
                FORMAT := 16#0000,
                P := 45,
                OUT => "SET VALUE"."SET HPHV UP T2");
   END_IF;
   VAL_STRG(IN := "new"."HPHV SET TEMP"[2],
            SIZE := 5,
            PREC := 1,
            FORMAT := 16#0000,
            P := 45,
            OUT => "SET VALUE"."SET HPHV HT3",
            ENO => #_w8);
   IF #_w8 THEN
       VAL_STRG(IN := "new"."HPHV SET TIME"[2],
                SIZE := 4,
                PREC := 0,
                FORMAT := 16#0000,
                P := 45,
                OUT => "SET VALUE"."SET HPHV UP T3");
   END_IF;
   VAL_STRG(IN := "new"."HPHV STOP TEMP",
            SIZE := 5,
            PREC := 1,
            FORMAT := 16#0000,
            P := 45,
            OUT => "SET VALUE"."SET HPHV STOP TMP",
            ENO => #_w9);
   IF #_w9 THEN
       VAL_STRG(IN := "new"."HPHV SET TIME"[3],
                SIZE := 4,
                PREC := 0,
                FORMAT := 16#0000,
                P := 45,
                OUT => "SET VALUE"."SET HPHV POST PULSES");
   END_IF;
END_REGION

REGION Network 26
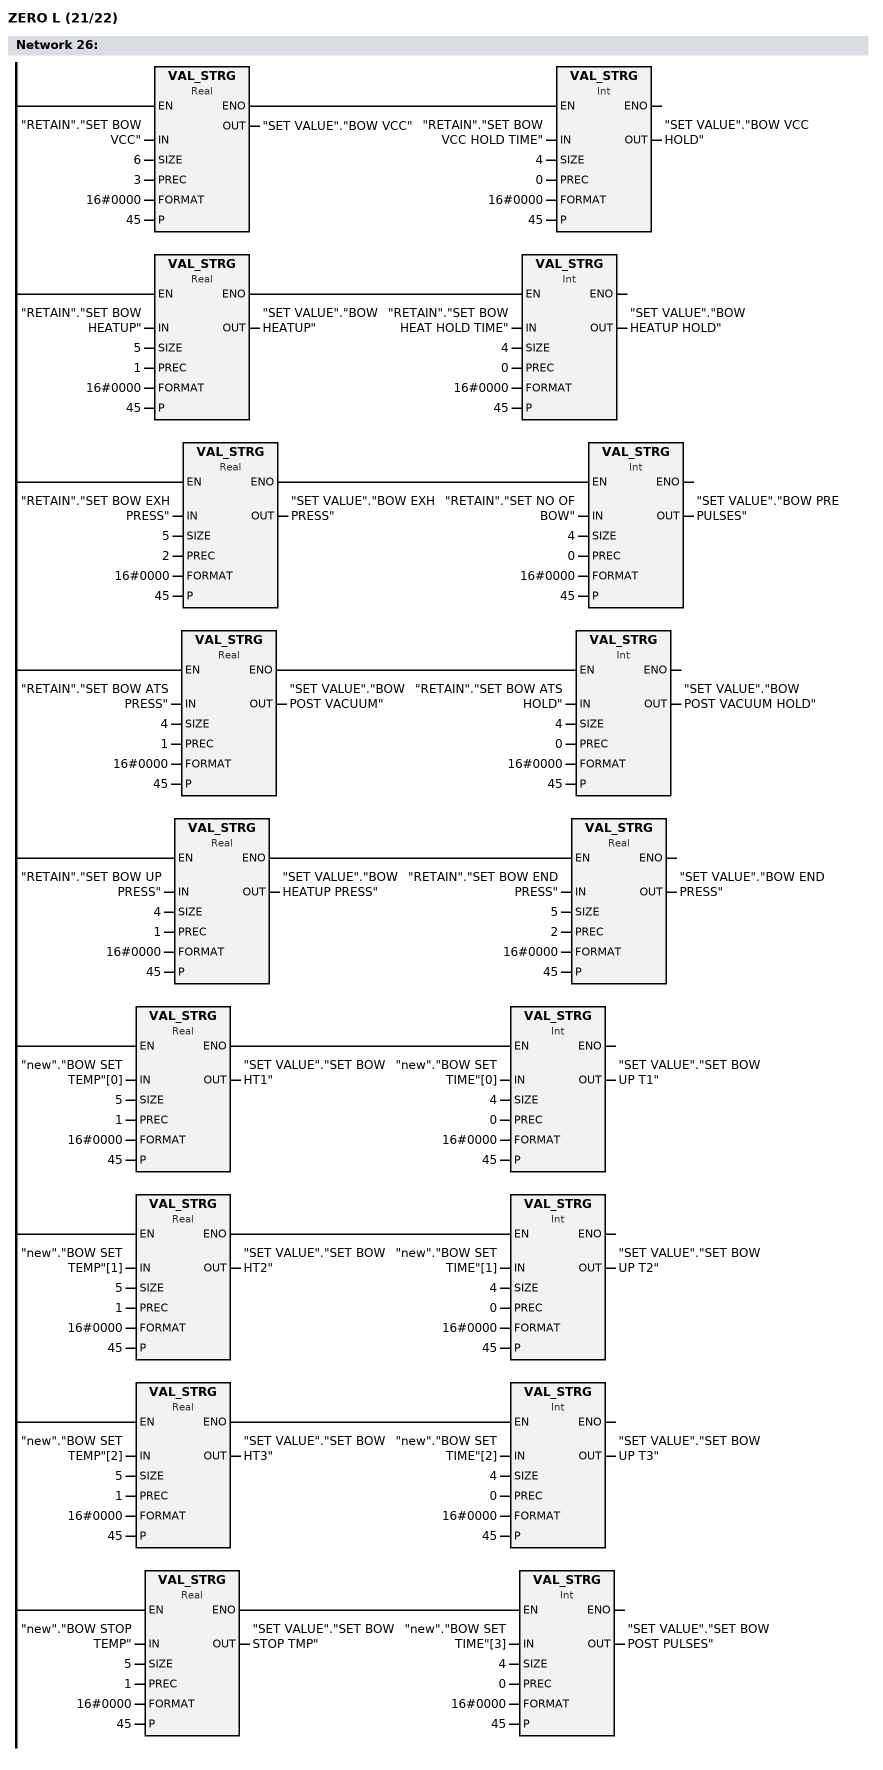
   RUNG wire#powerrail
      { S7_Templates := "[value_type := Real, str_type := String]" } VAL_STRG(IN := "RETAIN"."SET BOW VCC", SIZE := 6, PREC := 3, FORMAT := 16#0000, P := 45, OUT => "SET VALUE"."BOW VCC")
      { S7_Templates := "[value_type := Int, str_type := String]" } VAL_STRG(IN := "RETAIN"."SET BOW  VCC HOLD TIME", SIZE := 4, PREC := 0, FORMAT := 16#0000, P := 45, OUT => "SET VALUE"."BOW VCC HOLD")
   END_RUNG
   RUNG wire#powerrail
      { S7_Templates := "[value_type := Real, str_type := String]" } VAL_STRG(IN := "RETAIN"."SET BOW HEATUP", SIZE := 5, PREC := 1, FORMAT := 16#0000, P := 45, OUT => "SET VALUE"."BOW HEATUP")
      { S7_Templates := "[value_type := Int, str_type := String]" } VAL_STRG(IN := "RETAIN"."SET BOW HEAT HOLD TIME", SIZE := 4, PREC := 0, FORMAT := 16#0000, P := 45, OUT => "SET VALUE"."BOW HEATUP HOLD")
   END_RUNG
   RUNG wire#powerrail
      { S7_Templates := "[value_type := Real, str_type := String]" } VAL_STRG(IN := "RETAIN"."SET BOW EXH PRESS", SIZE := 5, PREC := 2, FORMAT := 16#0000, P := 45, OUT => "SET VALUE"."BOW EXH PRESS")
      { S7_Templates := "[value_type := Int, str_type := String]" } VAL_STRG(IN := "RETAIN"."SET NO OF BOW", SIZE := 4, PREC := 0, FORMAT := 16#0000, P := 45, OUT => "SET VALUE"."BOW PRE PULSES")
   END_RUNG
   RUNG wire#powerrail
      { S7_Templates := "[value_type := Real, str_type := String]" } VAL_STRG(IN := "RETAIN"."SET BOW ATS PRESS", SIZE := 4, PREC := 1, FORMAT := 16#0000, P := 45, OUT => "SET VALUE"."BOW POST VACUUM")
      { S7_Templates := "[value_type := Int, str_type := String]" } VAL_STRG(IN := "RETAIN"."SET BOW ATS HOLD", SIZE := 4, PREC := 0, FORMAT := 16#0000, P := 45, OUT => "SET VALUE"."BOW POST VACUUM HOLD")
   END_RUNG
   RUNG wire#powerrail
      { S7_Templates := "[value_type := Real, str_type := String]" } VAL_STRG(IN := "RETAIN"."SET BOW UP PRESS", SIZE := 4, PREC := 1, FORMAT := 16#0000, P := 45, OUT => "SET VALUE"."BOW HEATUP PRESS")
      { S7_Templates := "[value_type := Real, str_type := String]" } VAL_STRG(IN := "RETAIN"."SET BOW END PRESS", SIZE := 5, PREC := 2, FORMAT := 16#0000, P := 45, OUT => "SET VALUE"."BOW END PRESS")
   END_RUNG
   RUNG wire#powerrail
      { S7_Templates := "[value_type := Real, str_type := String]" } VAL_STRG(IN := "new"."BOW SET TEMP"[0], SIZE := 5, PREC := 1, FORMAT := 16#0000, P := 45, OUT => "SET VALUE"."SET BOW HT1")
      { S7_Templates := "[value_type := Int, str_type := String]" } VAL_STRG(IN := "new"."BOW SET TIME"[0], SIZE := 4, PREC := 0, FORMAT := 16#0000, P := 45, OUT => "SET VALUE"."SET BOW UP T1")
   END_RUNG
   RUNG wire#powerrail
      { S7_Templates := "[value_type := Real, str_type := String]" } VAL_STRG(IN := "new"."BOW SET TEMP"[1], SIZE := 5, PREC := 1, FORMAT := 16#0000, P := 45, OUT => "SET VALUE"."SET BOW HT2")
      { S7_Templates := "[value_type := Int, str_type := String]" } VAL_STRG(IN := "new"."BOW SET TIME"[1], SIZE := 4, PREC := 0, FORMAT := 16#0000, P := 45, OUT => "SET VALUE"."SET BOW UP T2")
   END_RUNG
   RUNG wire#powerrail
      { S7_Templates := "[value_type := Real, str_type := String]" } VAL_STRG(IN := "new"."BOW SET TEMP"[2], SIZE := 5, PREC := 1, FORMAT := 16#0000, P := 45, OUT => "SET VALUE"."SET BOW HT3")
      { S7_Templates := "[value_type := Int, str_type := String]" } VAL_STRG(IN := "new"."BOW SET TIME"[2], SIZE := 4, PREC := 0, FORMAT := 16#0000, P := 45, OUT => "SET VALUE"."SET BOW UP T3")
   END_RUNG
   RUNG wire#powerrail
      { S7_Templates := "[value_type := Real, str_type := String]" } VAL_STRG(IN := "new"."BOW STOP TEMP", SIZE := 5, PREC := 1, FORMAT := 16#0000, P := 45, OUT => "SET VALUE"."SET BOW STOP TMP")
      { S7_Templates := "[value_type := Int, str_type := String]" } VAL_STRG(IN := "new"."BOW SET TIME"[3], SIZE := 4, PREC := 0, FORMAT := 16#0000, P := 45, OUT => "SET VALUE"."SET BOW POST PULSES")
   END_RUNG
   // the same network as SCL:
   VAL_STRG(IN := "RETAIN"."SET BOW VCC",
            SIZE := 6,
            PREC := 3,
            FORMAT := 16#0000,
            P := 45,
            OUT => "SET VALUE"."BOW VCC",
            ENO => #_w1);
   IF #_w1 THEN
       VAL_STRG(IN := "RETAIN"."SET BOW  VCC HOLD TIME",
                SIZE := 4,
                PREC := 0,
                FORMAT := 16#0000,
                P := 45,
                OUT => "SET VALUE"."BOW VCC HOLD");
   END_IF;
   VAL_STRG(IN := "RETAIN"."SET BOW HEATUP",
            SIZE := 5,
            PREC := 1,
            FORMAT := 16#0000,
            P := 45,
            OUT => "SET VALUE"."BOW HEATUP",
            ENO => #_w2);
   IF #_w2 THEN
       VAL_STRG(IN := "RETAIN"."SET BOW HEAT HOLD TIME",
                SIZE := 4,
                PREC := 0,
                FORMAT := 16#0000,
                P := 45,
                OUT => "SET VALUE"."BOW HEATUP HOLD");
   END_IF;
   VAL_STRG(IN := "RETAIN"."SET BOW EXH PRESS",
            SIZE := 5,
            PREC := 2,
            FORMAT := 16#0000,
            P := 45,
            OUT => "SET VALUE"."BOW EXH PRESS",
            ENO => #_w3);
   IF #_w3 THEN
       VAL_STRG(IN := "RETAIN"."SET NO OF BOW",
                SIZE := 4,
                PREC := 0,
                FORMAT := 16#0000,
                P := 45,
                OUT => "SET VALUE"."BOW PRE PULSES");
   END_IF;
   VAL_STRG(IN := "RETAIN"."SET BOW ATS PRESS",
            SIZE := 4,
            PREC := 1,
            FORMAT := 16#0000,
            P := 45,
            OUT => "SET VALUE"."BOW POST VACUUM",
            ENO => #_w4);
   IF #_w4 THEN
       VAL_STRG(IN := "RETAIN"."SET BOW ATS HOLD",
                SIZE := 4,
                PREC := 0,
                FORMAT := 16#0000,
                P := 45,
                OUT => "SET VALUE"."BOW POST VACUUM HOLD");
   END_IF;
   VAL_STRG(IN := "RETAIN"."SET BOW UP PRESS",
            SIZE := 4,
            PREC := 1,
            FORMAT := 16#0000,
            P := 45,
            OUT => "SET VALUE"."BOW HEATUP PRESS",
            ENO => #_w5);
   IF #_w5 THEN
       VAL_STRG(IN := "RETAIN"."SET BOW END PRESS",
                SIZE := 5,
                PREC := 2,
                FORMAT := 16#0000,
                P := 45,
                OUT => "SET VALUE"."BOW END PRESS");
   END_IF;
   VAL_STRG(IN := "new"."BOW SET TEMP"[0],
            SIZE := 5,
            PREC := 1,
            FORMAT := 16#0000,
            P := 45,
            OUT => "SET VALUE"."SET BOW HT1",
            ENO => #_w6);
   IF #_w6 THEN
       VAL_STRG(IN := "new"."BOW SET TIME"[0],
                SIZE := 4,
                PREC := 0,
                FORMAT := 16#0000,
                P := 45,
                OUT => "SET VALUE"."SET BOW UP T1");
   END_IF;
   VAL_STRG(IN := "new"."BOW SET TEMP"[1],
            SIZE := 5,
            PREC := 1,
            FORMAT := 16#0000,
            P := 45,
            OUT => "SET VALUE"."SET BOW HT2",
            ENO => #_w7);
   IF #_w7 THEN
       VAL_STRG(IN := "new"."BOW SET TIME"[1],
                SIZE := 4,
                PREC := 0,
                FORMAT := 16#0000,
                P := 45,
                OUT => "SET VALUE"."SET BOW UP T2");
   END_IF;
   VAL_STRG(IN := "new"."BOW SET TEMP"[2],
            SIZE := 5,
            PREC := 1,
            FORMAT := 16#0000,
            P := 45,
            OUT => "SET VALUE"."SET BOW HT3",
            ENO => #_w8);
   IF #_w8 THEN
       VAL_STRG(IN := "new"."BOW SET TIME"[2],
                SIZE := 4,
                PREC := 0,
                FORMAT := 16#0000,
                P := 45,
                OUT => "SET VALUE"."SET BOW UP T3");
   END_IF;
   VAL_STRG(IN := "new"."BOW STOP TEMP",
            SIZE := 5,
            PREC := 1,
            FORMAT := 16#0000,
            P := 45,
            OUT => "SET VALUE"."SET BOW STOP TMP",
            ENO => #_w9);
   IF #_w9 THEN
       VAL_STRG(IN := "new"."BOW SET TIME"[3],
                SIZE := 4,
                PREC := 0,
                FORMAT := 16#0000,
                P := 45,
                OUT => "SET VALUE"."SET BOW POST PULSES");
   END_IF;
END_REGION

REGION Network 27
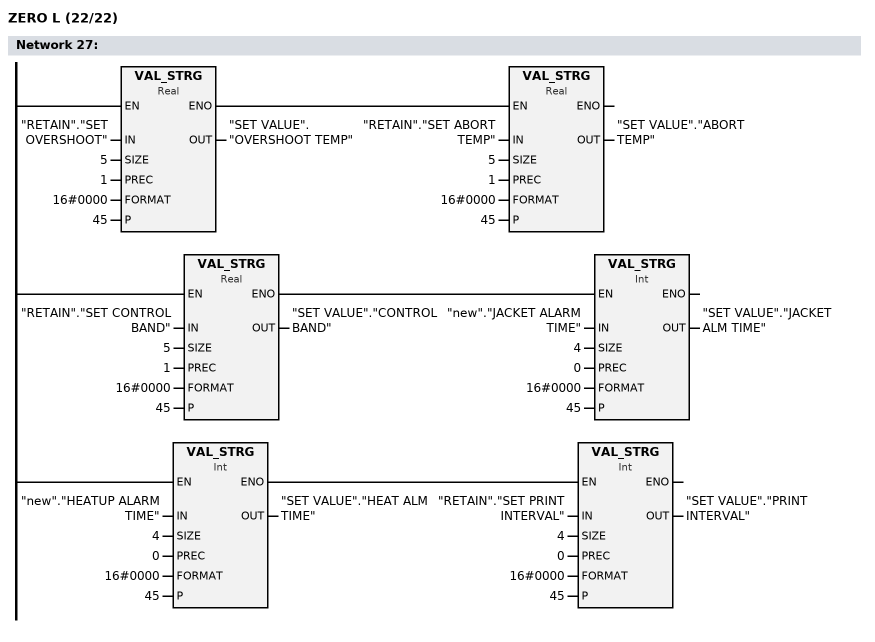
   RUNG wire#powerrail
      { S7_Templates := "[value_type := Real, str_type := String]" } VAL_STRG(IN := "RETAIN"."SET OVERSHOOT", SIZE := 5, PREC := 1, FORMAT := 16#0000, P := 45, OUT => "SET VALUE"."OVERSHOOT TEMP")
      { S7_Templates := "[value_type := Real, str_type := String]" } VAL_STRG(IN := "RETAIN"."SET ABORT TEMP", SIZE := 5, PREC := 1, FORMAT := 16#0000, P := 45, OUT => "SET VALUE"."ABORT TEMP")
   END_RUNG
   RUNG wire#powerrail
      { S7_Templates := "[value_type := Real, str_type := String]" } VAL_STRG(IN := "RETAIN"."SET CONTROL BAND", SIZE := 5, PREC := 1, FORMAT := 16#0000, P := 45, OUT => "SET VALUE"."CONTROL BAND")
      { S7_Templates := "[value_type := Int, str_type := String]" } VAL_STRG(IN := "new"."JACKET ALARM TIME", SIZE := 4, PREC := 0, FORMAT := 16#0000, P := 45, OUT => "SET VALUE"."JACKET ALM TIME")
   END_RUNG
   RUNG wire#powerrail
      { S7_Templates := "[value_type := Int, str_type := String]" } VAL_STRG(IN := "new"."HEATUP ALARM TIME", SIZE := 4, PREC := 0, FORMAT := 16#0000, P := 45, OUT => "SET VALUE"."HEAT ALM TIME")
      { S7_Templates := "[value_type := Int, str_type := String]" } VAL_STRG(IN := "RETAIN"."SET PRINT INTERVAL", SIZE := 4, PREC := 0, FORMAT := 16#0000, P := 45, OUT => "SET VALUE"."PRINT INTERVAL")
   END_RUNG
   // the same network as SCL:
   VAL_STRG(IN := "RETAIN"."SET OVERSHOOT",
            SIZE := 5,
            PREC := 1,
            FORMAT := 16#0000,
            P := 45,
            OUT => "SET VALUE"."OVERSHOOT TEMP",
            ENO => #_w1);
   IF #_w1 THEN
       VAL_STRG(IN := "RETAIN"."SET ABORT TEMP",
                SIZE := 5,
                PREC := 1,
                FORMAT := 16#0000,
                P := 45,
                OUT => "SET VALUE"."ABORT TEMP");
   END_IF;
   VAL_STRG(IN := "RETAIN"."SET CONTROL BAND",
            SIZE := 5,
            PREC := 1,
            FORMAT := 16#0000,
            P := 45,
            OUT => "SET VALUE"."CONTROL BAND",
            ENO => #_w2);
   IF #_w2 THEN
       VAL_STRG(IN := "new"."JACKET ALARM TIME",
                SIZE := 4,
                PREC := 0,
                FORMAT := 16#0000,
                P := 45,
                OUT => "SET VALUE"."JACKET ALM TIME");
   END_IF;
   VAL_STRG(IN := "new"."HEATUP ALARM TIME",
            SIZE := 4,
            PREC := 0,
            FORMAT := 16#0000,
            P := 45,
            OUT => "SET VALUE"."HEAT ALM TIME",
            ENO => #_w3);
   IF #_w3 THEN
       VAL_STRG(IN := "RETAIN"."SET PRINT INTERVAL",
                SIZE := 4,
                PREC := 0,
                FORMAT := 16#0000,
                P := 45,
                OUT => "SET VALUE"."PRINT INTERVAL");
   END_IF;
END_REGION
END_FUNCTION
